LIN {X 0,Y 466.491,Z 652.582,A -85,B 0,C 180,E1 -7510.377,E2 -7510.377} C_VEL
LIN {X 0,Y 466.525,Z 652.204,A -85,B 0,C 180,E1 -7511.517,E2 -7511.517} C_VEL
LIN {X 0,Y 466.577,Z 651.333,A -85,B 0,C 180,E1 -7512.674,E2 -7512.674} C_VEL
LIN {X 0,Y 466.638,Z 649.94,A -85,B 0,C 180,E1 -7513.852,E2 -7513.852} C_VEL
LIN {X 0,Y 466.788,Z 646.773,A -85,B 0,C 180,E1 -7515.615,E2 -7515.615} C_VEL
LIN {X 0,Y 466.978,Z 641.957,A -85,B 0,C 180,E1 -7517.514,E2 -7517.514} C_VEL
LIN {X 0,Y 467.197,Z 636.151,A -85,B 0,C 180,E1 -7519.246,E2 -7519.246} C_VEL
LIN {X 0,Y 467.651,Z 629.363,A -85,B 0,C 180,E1 -7520.861,E2 -7520.861} C_VEL
LIN {X 0,Y 468.11,Z 621.588,A -85,B 0,C 180,E1 -7522.389,E2 -7522.389} C_VEL
LIN {X 0,Y 468.72,Z 612.47,A -85,B 0,C 180,E1 -7523.882,E2 -7523.882} C_VEL
LIN {X 0,Y 469.512,Z 601.824,A -85,B 0,C 180,E1 -7525.332,E2 -7525.332} C_VEL
LIN {X 0,Y 470.362,Z 590.164,A -85,B 0,C 180,E1 -7526.653,E2 -7526.653} C_VEL
LIN {X 0,Y 471.18,Z 578.051,A -85,B 0,C 180,E1 -7527.796,E2 -7527.796} C_VEL
LIN {X 0,Y 472.008,Z 565.223,A -85,B 0,C 180,E1 -7528.797,E2 -7528.797} C_VEL
LIN {X 0,Y 472.783,Z 551.153,A -85,B 0,C 180,E1 -7529.687,E2 -7529.687} C_VEL
LIN {X 0,Y 473.449,Z 536.973,A -85,B 0,C 180,E1 -7530.392,E2 -7530.392} C_VEL
LIN {X 0,Y 473.761,Z 524.414,A -85,B 0,C 180,E1 -7530.885,E2 -7530.885} C_VEL
LIN {X 0,Y 471.201,Z 515.269,A -85,B 0,C 180,E1 -7531.292,E2 -7531.292} C_VEL
LIN {X 0,Y 467.058,Z 503.621,A -85,B 0,C 180,E1 -7531.767,E2 -7531.767} C_VEL
LIN {X 0,Y 466.908,Z 502.739,A -85,B 0,C 180,E1 -7531.818,E2 -7531.818} C_VEL
LIN {X 0,Y 467.035,Z 499.956,A -85,B 0,C 180,E1 -7535.08,E2 -7535.08} C_VEL
LIN {X 0,Y 467.083,Z 497.603,A -85,B 0,C 180,E1 -7537.903,E2 -7537.903} C_VEL
LIN {X 0,Y 467.194,Z 495.312,A -85,B 0,C 180,E1 -7540.673,E2 -7540.673} C_VEL
LIN {X 0,Y 467.284,Z 493.077,A -85,B 0,C 180,E1 -7543.395,E2 -7543.395} C_VEL
LIN {X 0,Y 467.325,Z 490.903,A -85,B 0,C 180,E1 -7546.076,E2 -7546.076} C_VEL
LIN {X 0,Y 467.611,Z 490.865,A -85,B 0,C 180,E1 -7548.732,E2 -7548.732} C_VEL
LIN {X 0,Y 467.746,Z 490.849,A -85,B 0,C 180,E1 -7552.228,E2 -7552.228} C_VEL
LIN {X 0,Y 467.724,Z 490.847,A -85,B 0,C 180,E1 -7554.827,E2 -7554.827} C_VEL
LIN {X 0,Y 467.857,Z 490.832,A -85,B 0,C 180,E1 -7557.417,E2 -7557.417} C_VEL
LIN {X 0,Y 467.878,Z 490.83,A -85,B 0,C 180,E1 -7560,E2 -7560} C_VEL
LIN {X 0,Y 467.856,Z 490.83,A -85,B 0,C 180,E1 -7562.583,E2 -7562.583} C_VEL
LIN {X 0,Y 467.744,Z 490.844,A -85,B 0,C 180,E1 -7566.037,E2 -7566.037} C_VEL
LIN {X 0,Y 467.678,Z 490.854,A -85,B 0,C 180,E1 -7568.643,E2 -7568.643} C_VEL
LIN {X 0,Y 467.653,Z 490.855,A -85,B 0,C 180,E1 -7572.145,E2 -7572.145} C_VEL
LIN {X 0,Y 467.635,Z 490.856,A -85,B 0,C 180,E1 -7575.695,E2 -7575.695} C_VEL
LIN {X 0,Y 467.614,Z 490.863,A -85,B 0,C 180,E1 -7578.765,E2 -7578.765} C_VEL
LIN {X 0,Y 467.577,Z 490.863,A -85,B 0,C 180,E1 -7581.268,E2 -7581.268} C_VEL
LIN {X 0,Y 467.57,Z 490.867,A -85,B 0,C 180,E1 -7583.943,E2 -7583.943} C_VEL
LIN {X 0,Y 467.624,Z 490.86,A -85,B 0,C 180,E1 -7586.8,E2 -7586.8} C_VEL
LIN {X 0,Y 467.584,Z 490.869,A -85,B 0,C 180,E1 -7589.736,E2 -7589.736} C_VEL
LIN {X 0,Y 467.581,Z 490.865,A -85,B 0,C 180,E1 -7592.758,E2 -7592.758} C_VEL
LIN {X 0,Y 467.554,Z 490.871,A -85,B 0,C 180,E1 -7595.889,E2 -7595.889} C_VEL
LIN {X 0,Y 467.579,Z 490.86,A -85,B 0,C 180,E1 -7599.145,E2 -7599.145} C_VEL
LIN {X 0,Y 467.599,Z 490.938,A -85,B 0,C 180,E1 -7602.267,E2 -7602.267} C_VEL
LIN {X 0,Y 468.484,Z 495.805,A -85,B 0,C 180,E1 -7605.165,E2 -7605.165} C_VEL
LIN {X 0,Y 469.206,Z 500.309,A -85,B 0,C 180,E1 -7607.621,E2 -7607.621} C_VEL
LIN {X 0,Y 469.155,Z 504.914,A -85,B 0,C 180,E1 -7609.899,E2 -7609.899} C_VEL
LIN {X 0,Y 468.717,Z 512.053,A -85,B 0,C 180,E1 -7613.147,E2 -7613.147} C_VEL
LIN {X 0,Y 468.459,Z 517.739,A -85,B 0,C 180,E1 -7615.601,E2 -7615.601} C_VEL
LIN {X 0,Y 468.157,Z 525.634,A -85,B 0,C 180,E1 -7618.835,E2 -7618.835} C_VEL
LIN {X 0,Y 467.78,Z 534.355,A -85,B 0,C 180,E1 -7622.241,E2 -7622.241} C_VEL
LIN {X 0,Y 467.603,Z 540.074,A -85,B 0,C 180,E1 -7624.394,E2 -7624.394} C_VEL
LIN {X 0,Y 467.385,Z 548.37,A -85,B 0,C 180,E1 -7627.453,E2 -7627.453} C_VEL
LIN {X 0,Y 467.349,Z 550.449,A -85,B 0,C 180,E1 -7628.204,E2 -7628.204} C_VEL
LIN {X 0,Y 471.32,Z 568.781,A -85,B 0,C 180,E1 -7628.795,E2 -7628.795} C_VEL
LIN {X 0,Y 473.467,Z 579.839,A -85,B 0,C 180,E1 -7629.253,E2 -7629.253} C_VEL
LIN {X 0,Y 472.829,Z 593.635,A -85,B 0,C 180,E1 -7629.807,E2 -7629.807} C_VEL
LIN {X 0,Y 472.025,Z 607.742,A -85,B 0,C 180,E1 -7630.54,E2 -7630.54} C_VEL
LIN {X 0,Y 471.223,Z 621.099,A -85,B 0,C 180,E1 -7631.41,E2 -7631.41} C_VEL
LIN {X 0,Y 470.317,Z 634.718,A -85,B 0,C 180,E1 -7632.498,E2 -7632.498} C_VEL
LIN {X 0,Y 469.526,Z 647.142,A -85,B 0,C 180,E1 -7633.701,E2 -7633.701} C_VEL
LIN {X 0,Y 468.759,Z 658.493,A -85,B 0,C 180,E1 -7635.011,E2 -7635.011} C_VEL
LIN {X 0,Y 468.082,Z 669.532,A -85,B 0,C 180,E1 -7636.542,E2 -7636.542} C_VEL
LIN {X 0,Y 467.594,Z 678.728,A -85,B 0,C 180,E1 -7638.073,E2 -7638.073} C_VEL
LIN {X 0,Y 467.244,Z 686.36,A -85,B 0,C 180,E1 -7639.601,E2 -7639.601} C_VEL
LIN {X 0,Y 466.954,Z 693.49,A -85,B 0,C 180,E1 -7641.343,E2 -7641.343} C_VEL
LIN {X 0,Y 466.819,Z 699.104,A -85,B 0,C 180,E1 -7643.082,E2 -7643.082} C_VEL
LIN {X 0,Y 466.718,Z 703.349,A -85,B 0,C 180,E1 -7644.816,E2 -7644.816} C_VEL
LIN {X 0,Y 466.724,Z 706.332,A -85,B 0,C 180,E1 -7646.546,E2 -7646.546} C_VEL
LIN {X 0,Y 466.681,Z 708.117,A -85,B 0,C 180,E1 -7648.274,E2 -7648.274} C_VEL
LIN {X 0,Y 466.595,Z 708.733,A -85,B 0,C 180,E1 -7650,E2 -7650} C_VEL
LIN {X 0,Y 466.681,Z 708.143,A -85,B 0,C 180,E1 -7651.725,E2 -7651.725} C_VEL
LIN {X 0,Y 466.705,Z 706.385,A -85,B 0,C 180,E1 -7653.453,E2 -7653.453} C_VEL
LIN {X 0,Y 466.717,Z 703.435,A -85,B 0,C 180,E1 -7655.183,E2 -7655.183} C_VEL
LIN {X 0,Y 466.816,Z 699.23,A -85,B 0,C 180,E1 -7656.917,E2 -7656.917} C_VEL
LIN {X 0,Y 466.953,Z 693.655,A -85,B 0,C 180,E1 -7658.656,E2 -7658.656} C_VEL
LIN {X 0,Y 467.243,Z 686.564,A -85,B 0,C 180,E1 -7660.398,E2 -7660.398} C_VEL
LIN {X 0,Y 467.584,Z 678.984,A -85,B 0,C 180,E1 -7661.927,E2 -7661.927} C_VEL
LIN {X 0,Y 468.089,Z 669.852,A -85,B 0,C 180,E1 -7663.457,E2 -7663.457} C_VEL
LIN {X 0,Y 468.792,Z 658.879,A -85,B 0,C 180,E1 -7664.987,E2 -7664.987} C_VEL
LIN {X 0,Y 469.6,Z 647.602,A -85,B 0,C 180,E1 -7666.296,E2 -7666.296} C_VEL
LIN {X 0,Y 470.395,Z 635.248,A -85,B 0,C 180,E1 -7667.498,E2 -7667.498} C_VEL
LIN {X 0,Y 471.333,Z 621.682,A -85,B 0,C 180,E1 -7668.585,E2 -7668.585} C_VEL
LIN {X 0,Y 472.069,Z 608.368,A -85,B 0,C 180,E1 -7669.457,E2 -7669.457} C_VEL
LIN {X 0,Y 472.884,Z 594.139,A -85,B 0,C 180,E1 -7670.199,E2 -7670.199} C_VEL
LIN {X 0,Y 473.519,Z 579.066,A -85,B 0,C 180,E1 -7670.8,E2 -7670.8} C_VEL
LIN {X 0,Y 470.319,Z 564.07,A -85,B 0,C 180,E1 -7671.388,E2 -7671.388} C_VEL
LIN {X 0,Y 467.41,Z 551.33,A -85,B 0,C 180,E1 -7671.791,E2 -7671.791} C_VEL
LIN {X 0,Y 467.633,Z 542.996,A -85,B 0,C 180,E1 -7674.885,E2 -7674.885} C_VEL
LIN {X 0,Y 467.969,Z 534.203,A -85,B 0,C 180,E1 -7678.233,E2 -7678.233} C_VEL
LIN {X 0,Y 468.238,Z 526.736,A -85,B 0,C 180,E1 -7681.181,E2 -7681.181} C_VEL
LIN {X 0,Y 468.555,Z 520.535,A -85,B 0,C 180,E1 -7683.708,E2 -7683.708} C_VEL
LIN {X 0,Y 468.964,Z 511.804,A -85,B 0,C 180,E1 -7687.414,E2 -7687.414} C_VEL
LIN {X 0,Y 469.354,Z 505.502,A -85,B 0,C 180,E1 -7690.212,E2 -7690.212} C_VEL
LIN {X 0,Y 469.457,Z 502.646,A -85,B 0,C 180,E1 -7691.538,E2 -7691.538} C_VEL
LIN {X 0,Y 468.984,Z 498.492,A -85,B 0,C 180,E1 -7693.576,E2 -7693.576} C_VEL
LIN {X 0,Y 468.021,Z 493.263,A -85,B 0,C 180,E1 -7696.31,E2 -7696.31} C_VEL
LIN {X 0,Y 467.608,Z 490.865,A -85,B 0,C 180,E1 -7697.661,E2 -7697.661} C_VEL
LIN {X 0,Y 467.616,Z 490.865,A -85,B 0,C 180,E1 -7700.859,E2 -7700.859} C_VEL
LIN {X 0,Y 467.554,Z 490.871,A -85,B 0,C 180,E1 -7704.26,E2 -7704.26} C_VEL
LIN {X 0,Y 467.573,Z 490.869,A -85,B 0,C 180,E1 -7707.32,E2 -7707.32} C_VEL
LIN {X 0,Y 467.569,Z 490.867,A -85,B 0,C 180,E1 -7710.665,E2 -7710.665} C_VEL
LIN {X 0,Y 467.618,Z 490.864,A -85,B 0,C 180,E1 -7713.2,E2 -7713.2} C_VEL
LIN {X 0,Y 467.582,Z 490.866,A -85,B 0,C 180,E1 -7716.468,E2 -7716.468} C_VEL
LIN {X 0,Y 467.614,Z 490.864,A -85,B 0,C 180,E1 -7719.777,E2 -7719.777} C_VEL
LIN {X 0,Y 467.599,Z 490.863,A -85,B 0,C 180,E1 -7722.507,E2 -7722.507} C_VEL
LIN {X 0,Y 467.596,Z 490.866,A -85,B 0,C 180,E1 -7725.196,E2 -7725.196} C_VEL
LIN {X 0,Y 467.672,Z 490.856,A -85,B 0,C 180,E1 -7727.855,E2 -7727.855} C_VEL
LIN {X 0,Y 467.673,Z 490.857,A -85,B 0,C 180,E1 -7731.357,E2 -7731.357} C_VEL
LIN {X 0,Y 467.738,Z 490.848,A -85,B 0,C 180,E1 -7733.963,E2 -7733.963} C_VEL
LIN {X 0,Y 467.852,Z 490.836,A -85,B 0,C 180,E1 -7737.417,E2 -7737.417} C_VEL
LIN {X 0,Y 467.872,Z 490.831,A -85,B 0,C 180,E1 -7740,E2 -7740} C_VEL
LIN {X 0,Y 467.853,Z 490.832,A -85,B 0,C 180,E1 -7742.583,E2 -7742.583} C_VEL
LIN {X 0,Y 467.745,Z 490.847,A -85,B 0,C 180,E1 -7746.038,E2 -7746.038} C_VEL
LIN {X 0,Y 467.673,Z 490.854,A -85,B 0,C 180,E1 -7748.643,E2 -7748.643} C_VEL
LIN {X 0,Y 467.647,Z 490.859,A -85,B 0,C 180,E1 -7752.146,E2 -7752.146} C_VEL
LIN {X 0,Y 467.63,Z 490.863,A -85,B 0,C 180,E1 -7755.696,E2 -7755.696} C_VEL
LIN {X 0,Y 467.609,Z 490.862,A -85,B 0,C 180,E1 -7758.766,E2 -7758.766} C_VEL
LIN {X 0,Y 467.572,Z 490.869,A -85,B 0,C 180,E1 -7761.269,E2 -7761.269} C_VEL
LIN {X 0,Y 467.565,Z 490.869,A -85,B 0,C 180,E1 -7763.944,E2 -7763.944} C_VEL
LIN {X 0,Y 467.62,Z 490.861,A -85,B 0,C 180,E1 -7766.801,E2 -7766.801} C_VEL
LIN {X 0,Y 467.581,Z 490.868,A -85,B 0,C 180,E1 -7769.737,E2 -7769.737} C_VEL
LIN {X 0,Y 467.578,Z 490.867,A -85,B 0,C 180,E1 -7772.759,E2 -7772.759} C_VEL
LIN {X 0,Y 467.551,Z 490.872,A -85,B 0,C 180,E1 -7775.89,E2 -7775.89} C_VEL
LIN {X 0,Y 467.619,Z 490.863,A -85,B 0,C 180,E1 -7779.142,E2 -7779.142} C_VEL
LIN {X 0,Y 467.615,Z 490.862,A -85,B 0,C 180,E1 -7782.573,E2 -7782.573} C_VEL
LIN {X 0,Y 467.571,Z 490.868,A -85,B 0,C 180,E1 -7786.178,E2 -7786.178} C_VEL
LIN {X 0,Y 467.588,Z 490.864,A -85,B 0,C 180,E1 -7788.723,E2 -7788.723} C_VEL
LIN {X 0,Y 467.577,Z 490.87,A -85,B 0,C 180,E1 -7791.408,E2 -7791.408} C_VEL
LIN {X 0,Y 467.562,Z 490.869,A -85,B 0,C 180,E1 -7794.262,E2 -7794.262} C_VEL
LIN {X 0,Y 467.582,Z 490.868,A -85,B 0,C 180,E1 -7797.322,E2 -7797.322} C_VEL
LIN {X 0,Y 467.571,Z 490.866,A -85,B 0,C 180,E1 -7800.668,E2 -7800.668} C_VEL
LIN {X 0,Y 467.63,Z 490.861,A -85,B 0,C 180,E1 -7803.202,E2 -7803.202} C_VEL
LIN {X 0,Y 467.595,Z 490.864,A -85,B 0,C 180,E1 -7806.469,E2 -7806.469} C_VEL
LIN {X 0,Y 467.626,Z 490.864,A -85,B 0,C 180,E1 -7809.778,E2 -7809.778} C_VEL
LIN {X 0,Y 467.613,Z 490.861,A -85,B 0,C 180,E1 -7812.508,E2 -7812.508} C_VEL
LIN {X 0,Y 467.601,Z 490.864,A -85,B 0,C 180,E1 -7815.434,E2 -7815.434} C_VEL
LIN {X 0,Y 466.931,Z 490.949,A -85,B 0,C 180,E1 -7816.153,E2 -7816.153} C_VEL
LIN {X 0,Y 464.087,Z 491.303,A -85,B 0,C 180,E1 -7817.322,E2 -7817.322} C_VEL
LIN {X 0,Y 461.687,Z 491.601,A -85,B 0,C 180,E1 -7818.264,E2 -7818.264} C_VEL
LIN {X 0,Y 460.66,Z 491.729,A -85,B 0,C 180,E1 -7818.991,E2 -7818.991} C_VEL
LIN {X 0,Y 460.578,Z 491.739,A -85,B 0,C 180,E1 -7819.238,E2 -7819.238} C_VEL
LIN {X 0,Y 460.693,Z 491.723,A -85,B 0,C 180,E1 -7822.57,E2 -7822.57} C_VEL
LIN {X 0,Y 460.703,Z 491.722,A -85,B 0,C 180,E1 -7824.749,E2 -7824.749} C_VEL
LIN {X 0,Y 460.83,Z 491.709,A -85,B 0,C 180,E1 -7827.378,E2 -7827.378} C_VEL
LIN {X 0,Y 460.858,Z 491.705,A -85,B 0,C 180,E1 -7830,E2 -7830} C_VEL
LIN {X 0,Y 460.594,Z 491.737,A -85,B 0,C 180,E1 -7832.624,E2 -7832.624} C_VEL
LIN {X 0,Y 460.297,Z 491.777,A -85,B 0,C 180,E1 -7835.257,E2 -7835.257} C_VEL
LIN {X 0,Y 460.121,Z 491.799,A -85,B 0,C 180,E1 -7836.138,E2 -7836.138} C_VEL
LIN {X 0,Y 460.102,Z 493.135,A -85,B 0,C 180,E1 -7837.902,E2 -7837.902} C_VEL
LIN {X 0,Y 460.014,Z 496.292,A -85,B 0,C 180,E1 -7841.456,E2 -7841.456} C_VEL
LIN {X 0,Y 459.909,Z 498.711,A -85,B 0,C 180,E1 -7844.152,E2 -7844.152} C_VEL
LIN {X 0,Y 459.833,Z 501.178,A -85,B 0,C 180,E1 -7846.882,E2 -7846.882} C_VEL
LIN {X 0,Y 459.829,Z 502.137,A -85,B 0,C 180,E1 -7847.937,E2 -7847.937} C_VEL
LIN {X 0,Y 461.465,Z 507.347,A -85,B 0,C 180,E1 -7848.146,E2 -7848.146} C_VEL
LIN {X 0,Y 466.199,Z 522.117,A -85,B 0,C 180,E1 -7848.791,E2 -7848.791} C_VEL
LIN {X 0,Y 467.154,Z 527.522,A -85,B 0,C 180,E1 -7849.032,E2 -7849.032} C_VEL
LIN {X 0,Y 466.486,Z 542.267,A -85,B 0,C 180,E1 -7849.656,E2 -7849.656} C_VEL
LIN {X 0,Y 465.662,Z 557.391,A -85,B 0,C 180,E1 -7850.499,E2 -7850.499} C_VEL
LIN {X 0,Y 464.865,Z 570.16,A -85,B 0,C 180,E1 -7851.391,E2 -7851.391} C_VEL
LIN {X 0,Y 464.098,Z 581.875,A -85,B 0,C 180,E1 -7852.378,E2 -7852.378} C_VEL
LIN {X 0,Y 463.162,Z 593.929,A -85,B 0,C 180,E1 -7853.591,E2 -7853.591} C_VEL
LIN {X 0,Y 462.346,Z 604.968,A -85,B 0,C 180,E1 -7854.926,E2 -7854.926} C_VEL
LIN {X 0,Y 461.592,Z 615.436,A -85,B 0,C 180,E1 -7856.446,E2 -7856.446} C_VEL
LIN {X 0,Y 461.007,Z 623.526,A -85,B 0,C 180,E1 -7857.845,E2 -7857.845} C_VEL
LIN {X 0,Y 460.468,Z 631.686,A -85,B 0,C 180,E1 -7859.543,E2 -7859.543} C_VEL
LIN {X 0,Y 460.087,Z 638.469,A -85,B 0,C 180,E1 -7861.289,E2 -7861.289} C_VEL
LIN {X 0,Y 459.855,Z 643.153,A -85,B 0,C 180,E1 -7862.799,E2 -7862.799} C_VEL
LIN {X 0,Y 459.702,Z 647.189,A -85,B 0,C 180,E1 -7864.448,E2 -7864.448} C_VEL
LIN {X 0,Y 459.529,Z 649.752,A -85,B 0,C 180,E1 -7865.847,E2 -7865.847} C_VEL
LIN {X 0,Y 459.456,Z 652.014,A -85,B 0,C 180,E1 -7867.723,E2 -7867.723} C_VEL
LIN {X 0,Y 459.446,Z 652.757,A -85,B 0,C 180,E1 -7868.841,E2 -7868.841} C_VEL
LIN {X 0,Y 459.408,Z 653.058,A -85,B 0,C 180,E1 -7870.101,E2 -7870.101} C_VEL
LIN {X 0,Y 459.437,Z 652.681,A -85,B 0,C 180,E1 -7871.448,E2 -7871.448} C_VEL
LIN {X 0,Y 459.507,Z 651.719,A -85,B 0,C 180,E1 -7872.764,E2 -7872.764} C_VEL
LIN {X 0,Y 459.61,Z 649.116,A -85,B 0,C 180,E1 -7874.7,E2 -7874.7} C_VEL
LIN {X 0,Y 459.799,Z 645.282,A -85,B 0,C 180,E1 -7876.541,E2 -7876.541} C_VEL
LIN {X 0,Y 460.021,Z 640.793,A -85,B 0,C 180,E1 -7878.149,E2 -7878.149} C_VEL
LIN {X 0,Y 460.286,Z 635.133,A -85,B 0,C 180,E1 -7879.768,E2 -7879.768} C_VEL
LIN {X 0,Y 460.697,Z 628.659,A -85,B 0,C 180,E1 -7881.283,E2 -7881.283} C_VEL
LIN {X 0,Y 461.331,Z 619.665,A -85,B 0,C 180,E1 -7883.004,E2 -7883.004} C_VEL
LIN {X 0,Y 461.987,Z 610.452,A -85,B 0,C 180,E1 -7884.465,E2 -7884.465} C_VEL
LIN {X 0,Y 462.822,Z 600.26,A -85,B 0,C 180,E1 -7885.816,E2 -7885.816} C_VEL
LIN {X 0,Y 463.639,Z 589.154,A -85,B 0,C 180,E1 -7887.057,E2 -7887.057} C_VEL
LIN {X 0,Y 464.497,Z 577.465,A -85,B 0,C 180,E1 -7888.151,E2 -7888.151} C_VEL
LIN {X 0,Y 465.314,Z 565.338,A -85,B 0,C 180,E1 -7889.1,E2 -7889.1} C_VEL
LIN {X 0,Y 466.128,Z 551.519,A -85,B 0,C 180,E1 -7889.983,E2 -7889.983} C_VEL
LIN {X 0,Y 466.839,Z 537.294,A -85,B 0,C 180,E1 -7890.698,E2 -7890.698} C_VEL
LIN {X 0,Y 467.137,Z 525.812,A -85,B 0,C 180,E1 -7891.159,E2 -7891.159} C_VEL
LIN {X 0,Y 464.156,Z 515.656,A -85,B 0,C 180,E1 -7891.636,E2 -7891.636} C_VEL
LIN {X 0,Y 459.868,Z 503.238,A -85,B 0,C 180,E1 -7892.165,E2 -7892.165} C_VEL
LIN {X 0,Y 459.963,Z 501.123,A -85,B 0,C 180,E1 -7894.67,E2 -7894.67} C_VEL
LIN {X 0,Y 460.028,Z 498.738,A -85,B 0,C 180,E1 -7897.546,E2 -7897.546} C_VEL
LIN {X 0,Y 460.118,Z 496.435,A -85,B 0,C 180,E1 -7900.364,E2 -7900.364} C_VEL
LIN {X 0,Y 460.217,Z 494.172,A -85,B 0,C 180,E1 -7903.133,E2 -7903.133} C_VEL
LIN {X 0,Y 460.28,Z 491.986,A -85,B 0,C 180,E1 -7905.859,E2 -7905.859} C_VEL
LIN {X 0,Y 460.557,Z 491.745,A -85,B 0,C 180,E1 -7908.558,E2 -7908.558} C_VEL
LIN {X 0,Y 460.626,Z 491.732,A -85,B 0,C 180,E1 -7911.223,E2 -7911.223} C_VEL
LIN {X 0,Y 460.708,Z 491.726,A -85,B 0,C 180,E1 -7913.87,E2 -7913.87} C_VEL
LIN {X 0,Y 460.822,Z 491.708,A -85,B 0,C 180,E1 -7917.377,E2 -7917.377} C_VEL
LIN {X 0,Y 460.849,Z 491.706,A -85,B 0,C 180,E1 -7920,E2 -7920} C_VEL
LIN {X 0,Y 460.821,Z 491.707,A -85,B 0,C 180,E1 -7922.622,E2 -7922.622} C_VEL
LIN {X 0,Y 460.709,Z 491.72,A -85,B 0,C 180,E1 -7926.13,E2 -7926.13} C_VEL
LIN {X 0,Y 460.625,Z 491.734,A -85,B 0,C 180,E1 -7928.776,E2 -7928.776} C_VEL
LIN {X 0,Y 460.609,Z 491.734,A -85,B 0,C 180,E1 -7932.445,E2 -7932.445} C_VEL
LIN {X 0,Y 460.596,Z 491.733,A -85,B 0,C 180,E1 -7935.997,E2 -7935.997} C_VEL
LIN {X 0,Y 460.567,Z 491.739,A -85,B 0,C 180,E1 -7938.902,E2 -7938.902} C_VEL
LIN {X 0,Y 460.512,Z 491.743,A -85,B 0,C 180,E1 -7941.485,E2 -7941.485} C_VEL
LIN {X 0,Y 460.539,Z 491.746,A -85,B 0,C 180,E1 -7944.332,E2 -7944.332} C_VEL
LIN {X 0,Y 460.58,Z 491.736,A -85,B 0,C 180,E1 -7947.243,E2 -7947.243} C_VEL
LIN {X 0,Y 460.524,Z 491.747,A -85,B 0,C 180,E1 -7950.239,E2 -7950.239} C_VEL
LIN {X 0,Y 460.526,Z 491.745,A -85,B 0,C 180,E1 -7953.325,E2 -7953.325} C_VEL
LIN {X 0,Y 460.476,Z 491.752,A -85,B 0,C 180,E1 -7956.529,E2 -7956.529} C_VEL
LIN {X 0,Y 460.542,Z 491.737,A -85,B 0,C 180,E1 -7958.898,E2 -7958.898} C_VEL
LIN {X 0,Y 460.54,Z 491.815,A -85,B 0,C 180,E1 -7961.854,E2 -7961.854} C_VEL
LIN {X 0,Y 461.312,Z 496.089,A -85,B 0,C 180,E1 -7964.491,E2 -7964.491} C_VEL
LIN {X 0,Y 462.21,Z 501.339,A -85,B 0,C 180,E1 -7967.465,E2 -7967.465} C_VEL
LIN {X 0,Y 462.224,Z 505.369,A -85,B 0,C 180,E1 -7969.485,E2 -7969.485} C_VEL
LIN {X 0,Y 461.786,Z 511.771,A -85,B 0,C 180,E1 -7972.5,E2 -7972.5} C_VEL
LIN {X 0,Y 461.467,Z 518.181,A -85,B 0,C 180,E1 -7975.326,E2 -7975.326} C_VEL
LIN {X 0,Y 461.118,Z 526.455,A -85,B 0,C 180,E1 -7978.788,E2 -7978.788} C_VEL
LIN {X 0,Y 460.733,Z 535.085,A -85,B 0,C 180,E1 -7982.218,E2 -7982.218} C_VEL
LIN {X 0,Y 460.489,Z 541.544,A -85,B 0,C 180,E1 -7984.701,E2 -7984.701} C_VEL
LIN {X 0,Y 460.288,Z 549.959,A -85,B 0,C 180,E1 -7987.848,E2 -7987.848} C_VEL
LIN {X 0,Y 464.082,Z 567.356,A -85,B 0,C 180,E1 -7988.424,E2 -7988.424} C_VEL
LIN {X 0,Y 466.744,Z 580.449,A -85,B 0,C 180,E1 -7988.982,E2 -7988.982} C_VEL
LIN {X 0,Y 466.081,Z 593.569,A -85,B 0,C 180,E1 -7989.524,E2 -7989.524} C_VEL
LIN {X 0,Y 465.29,Z 607.238,A -85,B 0,C 180,E1 -7990.247,E2 -7990.247} C_VEL
LIN {X 0,Y 464.444,Z 620.597,A -85,B 0,C 180,E1 -7991.128,E2 -7991.128} C_VEL
LIN {X 0,Y 463.472,Z 634.221,A -85,B 0,C 180,E1 -7992.231,E2 -7992.231} C_VEL
LIN {X 0,Y 462.655,Z 646.65,A -85,B 0,C 180,E1 -7993.452,E2 -7993.452} C_VEL
LIN {X 0,Y 461.814,Z 658,A -85,B 0,C 180,E1 -7994.781,E2 -7994.781} C_VEL
LIN {X 0,Y 461.095,Z 669.045,A -85,B 0,C 180,E1 -7996.334,E2 -7996.334} C_VEL
LIN {X 0,Y 460.535,Z 678.247,A -85,B 0,C 180,E1 -7997.887,E2 -7997.887} C_VEL
LIN {X 0,Y 460.175,Z 685.89,A -85,B 0,C 180,E1 -7999.439,E2 -7999.439} C_VEL
LIN {X 0,Y 459.888,Z 693.032,A -85,B 0,C 180,E1 -8001.209,E2 -8001.209} C_VEL
LIN {X 0,Y 459.729,Z 698.654,A -85,B 0,C 180,E1 -8002.975,E2 -8002.975} C_VEL
LIN {X 0,Y 459.626,Z 702.908,A -85,B 0,C 180,E1 -8004.736,E2 -8004.736} C_VEL
LIN {X 0,Y 459.633,Z 705.898,A -85,B 0,C 180,E1 -8006.493,E2 -8006.493} C_VEL
LIN {X 0,Y 459.616,Z 707.688,A -85,B 0,C 180,E1 -8008.247,E2 -8008.247} C_VEL
LIN {X 0,Y 459.527,Z 708.309,A -85,B 0,C 180,E1 -8010,E2 -8010} C_VEL
LIN {X 0,Y 459.616,Z 707.721,A -85,B 0,C 180,E1 -8011.752,E2 -8011.752} C_VEL
LIN {X 0,Y 459.617,Z 705.963,A -85,B 0,C 180,E1 -8013.506,E2 -8013.506} C_VEL
LIN {X 0,Y 459.626,Z 703.013,A -85,B 0,C 180,E1 -8015.263,E2 -8015.263} C_VEL
LIN {X 0,Y 459.727,Z 698.806,A -85,B 0,C 180,E1 -8017.024,E2 -8017.024} C_VEL
LIN {X 0,Y 459.887,Z 693.229,A -85,B 0,C 180,E1 -8018.79,E2 -8018.79} C_VEL
LIN {X 0,Y 460.173,Z 686.135,A -85,B 0,C 180,E1 -8020.56,E2 -8020.56} C_VEL
LIN {X 0,Y 460.536,Z 678.552,A -85,B 0,C 180,E1 -8022.112,E2 -8022.112} C_VEL
LIN {X 0,Y 461.103,Z 669.419,A -85,B 0,C 180,E1 -8023.664,E2 -8023.664} C_VEL
LIN {X 0,Y 461.828,Z 658.44,A -85,B 0,C 180,E1 -8025.218,E2 -8025.218} C_VEL
LIN {X 0,Y 462.697,Z 647.161,A -85,B 0,C 180,E1 -8026.546,E2 -8026.546} C_VEL
LIN {X 0,Y 463.534,Z 634.802,A -85,B 0,C 180,E1 -8027.765,E2 -8027.765} C_VEL
LIN {X 0,Y 464.525,Z 621.222,A -85,B 0,C 180,E1 -8028.867,E2 -8028.867} C_VEL
LIN {X 0,Y 465.35,Z 607.898,A -85,B 0,C 180,E1 -8029.749,E2 -8029.749} C_VEL
LIN {X 0,Y 466.167,Z 594.09,A -85,B 0,C 180,E1 -8030.48,E2 -8030.48} C_VEL
LIN {X 0,Y 466.68,Z 579.68,A -85,B 0,C 180,E1 -8031.076,E2 -8031.076} C_VEL
LIN {X 0,Y 463.342,Z 563.977,A -85,B 0,C 180,E1 -8031.713,E2 -8031.713} C_VEL
LIN {X 0,Y 460.364,Z 550.917,A -85,B 0,C 180,E1 -8032.141,E2 -8032.141} C_VEL
LIN {X 0,Y 460.623,Z 542.565,A -85,B 0,C 180,E1 -8035.29,E2 -8035.29} C_VEL
LIN {X 0,Y 460.958,Z 533.877,A -85,B 0,C 180,E1 -8038.702,E2 -8038.702} C_VEL
LIN {X 0,Y 461.264,Z 527.064,A -85,B 0,C 180,E1 -8041.435,E2 -8041.435} C_VEL
LIN {X 0,Y 461.577,Z 520.241,A -85,B 0,C 180,E1 -8044.287,E2 -8044.287} C_VEL
LIN {X 0,Y 462.007,Z 512.325,A -85,B 0,C 180,E1 -8047.72,E2 -8047.72} C_VEL
LIN {X 0,Y 462.423,Z 505.546,A -85,B 0,C 180,E1 -8050.806,E2 -8050.806} C_VEL
LIN {X 0,Y 462.348,Z 501.938,A -85,B 0,C 180,E1 -8052.536,E2 -8052.536} C_VEL
LIN {X 0,Y 461.349,Z 496.199,A -85,B 0,C 180,E1 -8055.513,E2 -8055.513} C_VEL
LIN {X 0,Y 460.562,Z 491.743,A -85,B 0,C 180,E1 -8057.985,E2 -8057.985} C_VEL
LIN {X 0,Y 460.541,Z 491.745,A -85,B 0,C 180,E1 -8061.269,E2 -8061.269} C_VEL
LIN {X 0,Y 460.505,Z 491.748,A -85,B 0,C 180,E1 -8064.554,E2 -8064.554} C_VEL
LIN {X 0,Y 460.523,Z 491.747,A -85,B 0,C 180,E1 -8067.715,E2 -8067.715} C_VEL
LIN {X 0,Y 460.538,Z 491.743,A -85,B 0,C 180,E1 -8070.769,E2 -8070.769} C_VEL
LIN {X 0,Y 460.558,Z 491.743,A -85,B 0,C 180,E1 -8073.735,E2 -8073.735} C_VEL
LIN {X 0,Y 460.536,Z 491.743,A -85,B 0,C 180,E1 -8076.624,E2 -8076.624} C_VEL
LIN {X 0,Y 460.542,Z 491.746,A -85,B 0,C 180,E1 -8079.453,E2 -8079.453} C_VEL
LIN {X 0,Y 460.549,Z 491.741,A -85,B 0,C 180,E1 -8082.23,E2 -8082.23} C_VEL
LIN {X 0,Y 460.559,Z 491.741,A -85,B 0,C 180,E1 -8084.965,E2 -8084.965} C_VEL
LIN {X 0,Y 460.619,Z 491.736,A -85,B 0,C 180,E1 -8087.666,E2 -8087.666} C_VEL
LIN {X 0,Y 460.62,Z 491.735,A -85,B 0,C 180,E1 -8091.224,E2 -8091.224} C_VEL
LIN {X 0,Y 460.703,Z 491.725,A -85,B 0,C 180,E1 -8093.87,E2 -8093.87} C_VEL
LIN {X 0,Y 460.817,Z 491.712,A -85,B 0,C 180,E1 -8097.378,E2 -8097.378} C_VEL
LIN {X 0,Y 460.843,Z 491.707,A -85,B 0,C 180,E1 -8100,E2 -8100} C_VEL
LIN {X 0,Y 460.818,Z 491.708,A -85,B 0,C 180,E1 -8102.623,E2 -8102.623} C_VEL
LIN {X 0,Y 460.709,Z 491.722,A -85,B 0,C 180,E1 -8106.13,E2 -8106.13} C_VEL
LIN {X 0,Y 460.62,Z 491.733,A -85,B 0,C 180,E1 -8108.777,E2 -8108.777} C_VEL
LIN {X 0,Y 460.603,Z 491.735,A -85,B 0,C 180,E1 -8112.446,E2 -8112.446} C_VEL
LIN {X 0,Y 460.591,Z 491.738,A -85,B 0,C 180,E1 -8115.998,E2 -8115.998} C_VEL
LIN {X 0,Y 460.562,Z 491.74,A -85,B 0,C 180,E1 -8118.903,E2 -8118.903} C_VEL
LIN {X 0,Y 460.508,Z 491.751,A -85,B 0,C 180,E1 -8121.486,E2 -8121.486} C_VEL
LIN {X 0,Y 460.535,Z 491.744,A -85,B 0,C 180,E1 -8124.333,E2 -8124.333} C_VEL
LIN {X 0,Y 460.577,Z 491.741,A -85,B 0,C 180,E1 -8127.244,E2 -8127.244} C_VEL
LIN {X 0,Y 460.52,Z 491.746,A -85,B 0,C 180,E1 -8130.24,E2 -8130.24} C_VEL
LIN {X 0,Y 460.523,Z 491.747,A -85,B 0,C 180,E1 -8133.326,E2 -8133.326} C_VEL
LIN {X 0,Y 460.474,Z 491.751,A -85,B 0,C 180,E1 -8136.53,E2 -8136.53} C_VEL
LIN {X 0,Y 460.58,Z 491.741,A -85,B 0,C 180,E1 -8139.858,E2 -8139.858} C_VEL
LIN {X 0,Y 460.539,Z 491.744,A -85,B 0,C 180,E1 -8142.906,E2 -8142.906} C_VEL
LIN {X 0,Y 460.521,Z 491.748,A -85,B 0,C 180,E1 -8145.83,E2 -8145.83} C_VEL
LIN {X 0,Y 460.541,Z 491.743,A -85,B 0,C 180,E1 -8148.991,E2 -8148.991} C_VEL
LIN {X 0,Y 460.546,Z 491.745,A -85,B 0,C 180,E1 -8151.27,E2 -8151.27} C_VEL
LIN {X 0,Y 460.512,Z 491.746,A -85,B 0,C 180,E1 -8154.556,E2 -8154.556} C_VEL
LIN {X 0,Y 460.532,Z 491.748,A -85,B 0,C 180,E1 -8157.717,E2 -8157.717} C_VEL
LIN {X 0,Y 460.541,Z 491.742,A -85,B 0,C 180,E1 -8160.77,E2 -8160.77} C_VEL
LIN {X 0,Y 460.57,Z 491.742,A -85,B 0,C 180,E1 -8163.736,E2 -8163.736} C_VEL
LIN {X 0,Y 460.549,Z 491.742,A -85,B 0,C 180,E1 -8166.625,E2 -8166.625} C_VEL
LIN {X 0,Y 460.554,Z 491.744,A -85,B 0,C 180,E1 -8169.454,E2 -8169.454} C_VEL
LIN {X 0,Y 460.563,Z 491.74,A -85,B 0,C 180,E1 -8172.231,E2 -8172.231} C_VEL
LIN {X 0,Y 460.57,Z 491.74,A -85,B 0,C 180,E1 -8174.966,E2 -8174.966} C_VEL
LIN {X 0,Y 460.614,Z 491.734,A -85,B 0,C 180,E1 -8178.56,E2 -8178.56} C_VEL
LIN {X 0,Y 460.578,Z 491.739,A -85,B 0,C 180,E1 -8179.238,E2 -8179.238} C_VEL
LIN {X 0,Y 459.919,Z 491.824,A -85,B 0,C 180,E1 -8179.968,E2 -8179.968} C_VEL
LIN {X 0,Y 457.091,Z 492.176,A -85,B 0,C 180,E1 -8181.154,E2 -8181.154} C_VEL
LIN {X 0,Y 454.708,Z 492.47,A -85,B 0,C 180,E1 -8182.11,E2 -8182.11} C_VEL
LIN {X 0,Y 453.7,Z 492.594,A -85,B 0,C 180,E1 -8182.849,E2 -8182.849} C_VEL
LIN {X 0,Y 453.627,Z 492.603,A -85,B 0,C 180,E1 -8183.099,E2 -8183.099} C_VEL
LIN {X 0,Y 453.676,Z 492.597,A -85,B 0,C 180,E1 -8184.667,E2 -8184.667} C_VEL
LIN {X 0,Y 453.771,Z 492.588,A -85,B 0,C 180,E1 -8187.337,E2 -8187.337} C_VEL
LIN {X 0,Y 453.828,Z 492.58,A -85,B 0,C 180,E1 -8190,E2 -8190} C_VEL
LIN {X 0,Y 453.551,Z 492.614,A -85,B 0,C 180,E1 -8192.665,E2 -8192.665} C_VEL
LIN {X 0,Y 453.236,Z 492.656,A -85,B 0,C 180,E1 -8195.339,E2 -8195.339} C_VEL
LIN {X 0,Y 453.069,Z 492.677,A -85,B 0,C 180,E1 -8196.234,E2 -8196.234} C_VEL
LIN {X 0,Y 453.027,Z 493.993,A -85,B 0,C 180,E1 -8198.026,E2 -8198.026} C_VEL
LIN {X 0,Y 452.944,Z 497.175,A -85,B 0,C 180,E1 -8201.637,E2 -8201.637} C_VEL
LIN {X 0,Y 452.833,Z 499.618,A -85,B 0,C 180,E1 -8204.378,E2 -8204.378} C_VEL
LIN {X 0,Y 452.767,Z 502.521,A -85,B 0,C 180,E1 -8207.59,E2 -8207.59} C_VEL
LIN {X 0,Y 455.296,Z 510.287,A -85,B 0,C 180,E1 -8207.895,E2 -8207.895} C_VEL
LIN {X 0,Y 459.894,Z 524.997,A -85,B 0,C 180,E1 -8208.575,E2 -8208.575} C_VEL
LIN {X 0,Y 460.502,Z 528.499,A -85,B 0,C 180,E1 -8208.742,E2 -8208.742} C_VEL
LIN {X 0,Y 459.773,Z 543.95,A -85,B 0,C 180,E1 -8209.418,E2 -8209.418} C_VEL
LIN {X 0,Y 459.036,Z 556.86,A -85,B 0,C 180,E1 -8210.15,E2 -8210.15} C_VEL
LIN {X 0,Y 458.161,Z 570.163,A -85,B 0,C 180,E1 -8211.083,E2 -8211.083} C_VEL
LIN {X 0,Y 457.325,Z 582.306,A -85,B 0,C 180,E1 -8212.118,E2 -8212.118} C_VEL
LIN {X 0,Y 456.317,Z 594.499,A -85,B 0,C 180,E1 -8213.365,E2 -8213.365} C_VEL
LIN {X 0,Y 455.516,Z 604.78,A -85,B 0,C 180,E1 -8214.618,E2 -8214.618} C_VEL
LIN {X 0,Y 454.695,Z 615.537,A -85,B 0,C 180,E1 -8216.191,E2 -8216.191} C_VEL
LIN {X 0,Y 454.031,Z 623.978,A -85,B 0,C 180,E1 -8217.67,E2 -8217.67} C_VEL
LIN {X 0,Y 453.445,Z 632.506,A -85,B 0,C 180,E1 -8219.478,E2 -8219.478} C_VEL
LIN {X 0,Y 453.02,Z 639.799,A -85,B 0,C 180,E1 -8221.432,E2 -8221.432} C_VEL
LIN {X 0,Y 452.77,Z 644.555,A -85,B 0,C 180,E1 -8223.048,E2 -8223.048} C_VEL
LIN {X 0,Y 452.56,Z 649.008,A -85,B 0,C 180,E1 -8225.071,E2 -8225.071} C_VEL
LIN {X 0,Y 452.432,Z 650.769,A -85,B 0,C 180,E1 -8226.177,E2 -8226.177} C_VEL
LIN {X 0,Y 452.378,Z 652.355,A -85,B 0,C 180,E1 -8227.596,E2 -8227.596} C_VEL
LIN {X 0,Y 452.343,Z 653.402,A -85,B 0,C 180,E1 -8229.569,E2 -8229.569} C_VEL
LIN {X 0,Y 452.324,Z 653.382,A -85,B 0,C 180,E1 -8230.736,E2 -8230.736} C_VEL
LIN {X 0,Y 452.354,Z 652.882,A -85,B 0,C 180,E1 -8231.918,E2 -8231.918} C_VEL
LIN {X 0,Y 452.436,Z 651.851,A -85,B 0,C 180,E1 -8233.116,E2 -8233.116} C_VEL
LIN {X 0,Y 452.577,Z 649.258,A -85,B 0,C 180,E1 -8234.955,E2 -8234.955} C_VEL
LIN {X 0,Y 452.798,Z 645.051,A -85,B 0,C 180,E1 -8236.926,E2 -8236.926} C_VEL
LIN {X 0,Y 453.027,Z 639.759,A -85,B 0,C 180,E1 -8238.751,E2 -8238.751} C_VEL
LIN {X 0,Y 453.49,Z 633.077,A -85,B 0,C 180,E1 -8240.55,E2 -8240.55} C_VEL
LIN {X 0,Y 453.973,Z 625.773,A -85,B 0,C 180,E1 -8242.142,E2 -8242.142} C_VEL
LIN {X 0,Y 454.697,Z 616.727,A -85,B 0,C 180,E1 -8243.774,E2 -8243.774} C_VEL
LIN {X 0,Y 455.429,Z 607.376,A -85,B 0,C 180,E1 -8245.182,E2 -8245.182} C_VEL
LIN {X 0,Y 456.345,Z 596.191,A -85,B 0,C 180,E1 -8246.593,E2 -8246.593} C_VEL
LIN {X 0,Y 457.267,Z 584.536,A -85,B 0,C 180,E1 -8247.819,E2 -8247.819} C_VEL
LIN {X 0,Y 458.187,Z 571.801,A -85,B 0,C 180,E1 -8248.935,E2 -8248.935} C_VEL
LIN {X 0,Y 459.089,Z 558.234,A -85,B 0,C 180,E1 -8249.905,E2 -8249.905} C_VEL
LIN {X 0,Y 459.962,Z 543.72,A -85,B 0,C 180,E1 -8250.728,E2 -8250.728} C_VEL
LIN {X 0,Y 460.602,Z 528.438,A -85,B 0,C 180,E1 -8251.392,E2 -8251.392} C_VEL
LIN {X 0,Y 459.381,Z 522.946,A -85,B 0,C 180,E1 -8251.657,E2 -8251.657} C_VEL
LIN {X 0,Y 454.635,Z 509.076,A -85,B 0,C 180,E1 -8252.307,E2 -8252.307} C_VEL
LIN {X 0,Y 452.848,Z 503.731,A -85,B 0,C 180,E1 -8252.534,E2 -8252.534} C_VEL
LIN {X 0,Y 452.913,Z 501.493,A -85,B 0,C 180,E1 -8255.23,E2 -8255.23} C_VEL
LIN {X 0,Y 453.036,Z 498.756,A -85,B 0,C 180,E1 -8258.556,E2 -8258.556} C_VEL
LIN {X 0,Y 453.124,Z 496.035,A -85,B 0,C 180,E1 -8261.928,E2 -8261.928} C_VEL
LIN {X 0,Y 453.243,Z 493.806,A -85,B 0,C 180,E1 -8264.716,E2 -8264.716} C_VEL
LIN {X 0,Y 453.299,Z 492.649,A -85,B 0,C 180,E1 -8266.552,E2 -8266.552} C_VEL
LIN {X 0,Y 453.507,Z 492.621,A -85,B 0,C 180,E1 -8269.282,E2 -8269.282} C_VEL
LIN {X 0,Y 453.689,Z 492.597,A -85,B 0,C 180,E1 -8272.48,E2 -8272.48} C_VEL
LIN {X 0,Y 453.67,Z 492.598,A -85,B 0,C 180,E1 -8274.666,E2 -8274.666} C_VEL
LIN {X 0,Y 453.763,Z 492.587,A -85,B 0,C 180,E1 -8277.336,E2 -8277.336} C_VEL
LIN {X 0,Y 453.82,Z 492.581,A -85,B 0,C 180,E1 -8280,E2 -8280} C_VEL
LIN {X 0,Y 453.761,Z 492.586,A -85,B 0,C 180,E1 -8282.663,E2 -8282.663} C_VEL
LIN {X 0,Y 453.676,Z 492.596,A -85,B 0,C 180,E1 -8286.225,E2 -8286.225} C_VEL
LIN {X 0,Y 453.589,Z 492.611,A -85,B 0,C 180,E1 -8288.913,E2 -8288.913} C_VEL
LIN {X 0,Y 453.559,Z 492.613,A -85,B 0,C 180,E1 -8292.529,E2 -8292.529} C_VEL
LIN {X 0,Y 453.541,Z 492.614,A -85,B 0,C 180,E1 -8296.196,E2 -8296.196} C_VEL
LIN {X 0,Y 453.516,Z 492.617,A -85,B 0,C 180,E1 -8299.041,E2 -8299.041} C_VEL
LIN {X 0,Y 453.473,Z 492.621,A -85,B 0,C 180,E1 -8301.836,E2 -8301.836} C_VEL
LIN {X 0,Y 453.511,Z 492.618,A -85,B 0,C 180,E1 -8304.734,E2 -8304.734} C_VEL
LIN {X 0,Y 453.535,Z 492.619,A -85,B 0,C 180,E1 -8307.961,E2 -8307.961} C_VEL
LIN {X 0,Y 453.48,Z 492.623,A -85,B 0,C 180,E1 -8310.759,E2 -8310.759} C_VEL
LIN {X 0,Y 453.475,Z 492.627,A -85,B 0,C 180,E1 -8313.913,E2 -8313.913} C_VEL
LIN {X 0,Y 453.468,Z 492.625,A -85,B 0,C 180,E1 -8317.188,E2 -8317.188} C_VEL
LIN {X 0,Y 453.487,Z 492.616,A -85,B 0,C 180,E1 -8319.45,E2 -8319.45} C_VEL
LIN {X 0,Y 453.516,Z 492.795,A -85,B 0,C 180,E1 -8321.489,E2 -8321.489} C_VEL
LIN {X 0,Y 454.405,Z 497.821,A -85,B 0,C 180,E1 -8324.647,E2 -8324.647} C_VEL
LIN {X 0,Y 455.171,Z 502.279,A -85,B 0,C 180,E1 -8327.206,E2 -8327.206} C_VEL
LIN {X 0,Y 455.28,Z 505.971,A -85,B 0,C 180,E1 -8329.147,E2 -8329.147} C_VEL
LIN {X 0,Y 454.783,Z 512.915,A -85,B 0,C 180,E1 -8332.468,E2 -8332.468} C_VEL
LIN {X 0,Y 454.48,Z 518.729,A -85,B 0,C 180,E1 -8335.099,E2 -8335.099} C_VEL
LIN {X 0,Y 454.133,Z 526.309,A -85,B 0,C 180,E1 -8338.338,E2 -8338.338} C_VEL
LIN {X 0,Y 453.755,Z 533.556,A -85,B 0,C 180,E1 -8341.305,E2 -8341.305} C_VEL
LIN {X 0,Y 453.487,Z 541.115,A -85,B 0,C 180,E1 -8344.282,E2 -8344.282} C_VEL
LIN {X 0,Y 453.251,Z 549.476,A -85,B 0,C 180,E1 -8347.48,E2 -8347.48} C_VEL
LIN {X 0,Y 457.234,Z 567.252,A -85,B 0,C 180,E1 -8348.09,E2 -8348.09} C_VEL
LIN {X 0,Y 459.971,Z 582.083,A -85,B 0,C 180,E1 -8348.739,E2 -8348.739} C_VEL
LIN {X 0,Y 459.305,Z 595.108,A -85,B 0,C 180,E1 -8349.314,E2 -8349.314} C_VEL
LIN {X 0,Y 458.442,Z 608.507,A -85,B 0,C 180,E1 -8350.056,E2 -8350.056} C_VEL
LIN {X 0,Y 457.549,Z 621.538,A -85,B 0,C 180,E1 -8350.949,E2 -8350.949} C_VEL
LIN {X 0,Y 456.524,Z 634.911,A -85,B 0,C 180,E1 -8352.068,E2 -8352.068} C_VEL
LIN {X 0,Y 455.748,Z 646.157,A -85,B 0,C 180,E1 -8353.193,E2 -8353.193} C_VEL
LIN {X 0,Y 454.872,Z 657.516,A -85,B 0,C 180,E1 -8354.542,E2 -8354.542} C_VEL
LIN {X 0,Y 454.122,Z 668.571,A -85,B 0,C 180,E1 -8356.12,E2 -8356.12} C_VEL
LIN {X 0,Y 453.49,Z 677.622,A -85,B 0,C 180,E1 -8357.668,E2 -8357.668} C_VEL
LIN {X 0,Y 453.136,Z 685.423,A -85,B 0,C 180,E1 -8359.274,E2 -8359.274} C_VEL
LIN {X 0,Y 452.794,Z 692.571,A -85,B 0,C 180,E1 -8361.07,E2 -8361.07} C_VEL
LIN {X 0,Y 452.648,Z 698.205,A -85,B 0,C 180,E1 -8362.864,E2 -8362.864} C_VEL
LIN {X 0,Y 452.538,Z 702.467,A -85,B 0,C 180,E1 -8364.653,E2 -8364.653} C_VEL
LIN {X 0,Y 452.531,Z 705.464,A -85,B 0,C 180,E1 -8366.438,E2 -8366.438} C_VEL
LIN {X 0,Y 452.523,Z 707.258,A -85,B 0,C 180,E1 -8368.22,E2 -8368.22} C_VEL
LIN {X 0,Y 452.461,Z 707.884,A -85,B 0,C 180,E1 -8370,E2 -8370} C_VEL
LIN {X 0,Y 452.523,Z 707.298,A -85,B 0,C 180,E1 -8371.779,E2 -8371.779} C_VEL
LIN {X 0,Y 452.516,Z 705.541,A -85,B 0,C 180,E1 -8373.561,E2 -8373.561} C_VEL
LIN {X 0,Y 452.538,Z 702.592,A -85,B 0,C 180,E1 -8375.346,E2 -8375.346} C_VEL
LIN {X 0,Y 452.646,Z 698.384,A -85,B 0,C 180,E1 -8377.135,E2 -8377.135} C_VEL
LIN {X 0,Y 452.81,Z 692.804,A -85,B 0,C 180,E1 -8378.928,E2 -8378.928} C_VEL
LIN {X 0,Y 453.135,Z 685.708,A -85,B 0,C 180,E1 -8380.726,E2 -8380.726} C_VEL
LIN {X 0,Y 453.512,Z 677.892,A -85,B 0,C 180,E1 -8382.345,E2 -8382.345} C_VEL
LIN {X 0,Y 454.138,Z 668.984,A -85,B 0,C 180,E1 -8383.878,E2 -8383.878} C_VEL
LIN {X 0,Y 454.89,Z 657.991,A -85,B 0,C 180,E1 -8385.456,E2 -8385.456} C_VEL
LIN {X 0,Y 455.77,Z 646.7,A -85,B 0,C 180,E1 -8386.805,E2 -8386.805} C_VEL
LIN {X 0,Y 456.709,Z 634.332,A -85,B 0,C 180,E1 -8388.04,E2 -8388.04} C_VEL
LIN {X 0,Y 457.71,Z 620.736,A -85,B 0,C 180,E1 -8389.159,E2 -8389.159} C_VEL
LIN {X 0,Y 458.618,Z 607.407,A -85,B 0,C 180,E1 -8390.052,E2 -8390.052} C_VEL
LIN {X 0,Y 459.511,Z 592.926,A -85,B 0,C 180,E1 -8390.825,E2 -8390.825} C_VEL
LIN {X 0,Y 459.925,Z 580.617,A -85,B 0,C 180,E1 -8391.344,E2 -8391.344} C_VEL
LIN {X 0,Y 456.533,Z 564.528,A -85,B 0,C 180,E1 -8392.024,E2 -8392.024} C_VEL
LIN {X 0,Y 453.298,Z 550.524,A -85,B 0,C 180,E1 -8392.493,E2 -8392.493} C_VEL
LIN {X 0,Y 453.612,Z 542.229,A -85,B 0,C 180,E1 -8395.709,E2 -8395.709} C_VEL
LIN {X 0,Y 453.898,Z 534.76,A -85,B 0,C 180,E1 -8398.684,E2 -8398.684} C_VEL
LIN {X 0,Y 454.242,Z 527.466,A -85,B 0,C 180,E1 -8401.685,E2 -8401.685} C_VEL
LIN {X 0,Y 454.574,Z 521.168,A -85,B 0,C 180,E1 -8404.353,E2 -8404.353} C_VEL
LIN {X 0,Y 455.043,Z 512.833,A -85,B 0,C 180,E1 -8408.031,E2 -8408.031} C_VEL
LIN {X 0,Y 455.44,Z 506.706,A -85,B 0,C 180,E1 -8410.876,E2 -8410.876} C_VEL
LIN {X 0,Y 455.32,Z 502.837,A -85,B 0,C 180,E1 -8412.776,E2 -8412.776} C_VEL
LIN {X 0,Y 454.271,Z 496.983,A -85,B 0,C 180,E1 -8415.878,E2 -8415.878} C_VEL
LIN {X 0,Y 453.515,Z 492.62,A -85,B 0,C 180,E1 -8418.362,E2 -8418.362} C_VEL
LIN {X 0,Y 453.527,Z 492.619,A -85,B 0,C 180,E1 -8420.786,E2 -8420.786} C_VEL
LIN {X 0,Y 453.449,Z 492.628,A -85,B 0,C 180,E1 -8423.917,E2 -8423.917} C_VEL
LIN {X 0,Y 453.474,Z 492.625,A -85,B 0,C 180,E1 -8427.151,E2 -8427.151} C_VEL
LIN {X 0,Y 453.505,Z 492.619,A -85,B 0,C 180,E1 -8430.271,E2 -8430.271} C_VEL
LIN {X 0,Y 453.504,Z 492.623,A -85,B 0,C 180,E1 -8433.294,E2 -8433.294} C_VEL
LIN {X 0,Y 453.493,Z 492.621,A -85,B 0,C 180,E1 -8436.239,E2 -8436.239} C_VEL
LIN {X 0,Y 453.473,Z 492.625,A -85,B 0,C 180,E1 -8439.117,E2 -8439.117} C_VEL
LIN {X 0,Y 453.502,Z 492.621,A -85,B 0,C 180,E1 -8441.944,E2 -8441.944} C_VEL
LIN {X 0,Y 453.539,Z 492.614,A -85,B 0,C 180,E1 -8444.727,E2 -8444.727} C_VEL
LIN {X 0,Y 453.591,Z 492.612,A -85,B 0,C 180,E1 -8447.472,E2 -8447.472} C_VEL
LIN {X 0,Y 453.584,Z 492.612,A -85,B 0,C 180,E1 -8451.087,E2 -8451.087} C_VEL
LIN {X 0,Y 453.67,Z 492.602,A -85,B 0,C 180,E1 -8453.775,E2 -8453.775} C_VEL
LIN {X 0,Y 453.758,Z 492.591,A -85,B 0,C 180,E1 -8457.337,E2 -8457.337} C_VEL
LIN {X 0,Y 453.814,Z 492.582,A -85,B 0,C 180,E1 -8460,E2 -8460} C_VEL
LIN {X 0,Y 453.758,Z 492.587,A -85,B 0,C 180,E1 -8462.664,E2 -8462.664} C_VEL
LIN {X 0,Y 453.675,Z 492.598,A -85,B 0,C 180,E1 -8466.226,E2 -8466.226} C_VEL
LIN {X 0,Y 453.584,Z 492.61,A -85,B 0,C 180,E1 -8468.914,E2 -8468.914} C_VEL
LIN {X 0,Y 453.554,Z 492.613,A -85,B 0,C 180,E1 -8472.53,E2 -8472.53} C_VEL
LIN {X 0,Y 453.536,Z 492.615,A -85,B 0,C 180,E1 -8476.197,E2 -8476.197} C_VEL
LIN {X 0,Y 453.512,Z 492.619,A -85,B 0,C 180,E1 -8479.042,E2 -8479.042} C_VEL
LIN {X 0,Y 453.468,Z 492.626,A -85,B 0,C 180,E1 -8481.837,E2 -8481.837} C_VEL
LIN {X 0,Y 453.507,Z 492.619,A -85,B 0,C 180,E1 -8484.735,E2 -8484.735} C_VEL
LIN {X 0,Y 453.532,Z 492.618,A -85,B 0,C 180,E1 -8487.962,E2 -8487.962} C_VEL
LIN {X 0,Y 453.477,Z 492.623,A -85,B 0,C 180,E1 -8490.76,E2 -8490.76} C_VEL
LIN {X 0,Y 453.472,Z 492.625,A -85,B 0,C 180,E1 -8493.914,E2 -8493.914} C_VEL
LIN {X 0,Y 453.467,Z 492.626,A -85,B 0,C 180,E1 -8497.189,E2 -8497.189} C_VEL
LIN {X 0,Y 453.532,Z 492.619,A -85,B 0,C 180,E1 -8499.446,E2 -8499.446} C_VEL
LIN {X 0,Y 453.488,Z 492.622,A -85,B 0,C 180,E1 -8502.993,E2 -8502.993} C_VEL
LIN {X 0,Y 453.474,Z 492.626,A -85,B 0,C 180,E1 -8505.782,E2 -8505.782} C_VEL
LIN {X 0,Y 453.494,Z 492.62,A -85,B 0,C 180,E1 -8508.213,E2 -8508.213} C_VEL
LIN {X 0,Y 453.531,Z 492.615,A -85,B 0,C 180,E1 -8510.789,E2 -8510.789} C_VEL
LIN {X 0,Y 453.456,Z 492.627,A -85,B 0,C 180,E1 -8513.919,E2 -8513.919} C_VEL
LIN {X 0,Y 453.483,Z 492.624,A -85,B 0,C 180,E1 -8517.152,E2 -8517.152} C_VEL
LIN {X 0,Y 453.476,Z 492.622,A -85,B 0,C 180,E1 -8520.27,E2 -8520.27} C_VEL
LIN {X 0,Y 453.516,Z 492.62,A -85,B 0,C 180,E1 -8523.296,E2 -8523.296} C_VEL
LIN {X 0,Y 453.506,Z 492.62,A -85,B 0,C 180,E1 -8526.24,E2 -8526.24} C_VEL
LIN {X 0,Y 453.486,Z 492.623,A -85,B 0,C 180,E1 -8529.119,E2 -8529.119} C_VEL
LIN {X 0,Y 453.516,Z 492.621,A -85,B 0,C 180,E1 -8531.946,E2 -8531.946} C_VEL
LIN {X 0,Y 453.544,Z 492.614,A -85,B 0,C 180,E1 -8534.727,E2 -8534.727} C_VEL
LIN {X 0,Y 453.563,Z 492.612,A -85,B 0,C 180,E1 -8538.38,E2 -8538.38} C_VEL
LIN {X 0,Y 453.59,Z 492.61,A -85,B 0,C 180,E1 -8541.087,E2 -8541.087} C_VEL
LIN {X 0,Y 453.627,Z 492.603,A -85,B 0,C 180,E1 -8543.099,E2 -8543.099} C_VEL
LIN {X 0,Y 452.951,Z 492.691,A -85,B 0,C 180,E1 -8543.84,E2 -8543.84} C_VEL
LIN {X 0,Y 450.009,Z 493.055,A -85,B 0,C 180,E1 -8545.041,E2 -8545.041} C_VEL
LIN {X 0,Y 447.587,Z 493.359,A -85,B 0,C 180,E1 -8546.011,E2 -8546.011} C_VEL
LIN {X 0,Y 446.65,Z 493.473,A -85,B 0,C 180,E1 -8546.761,E2 -8546.761} C_VEL
LIN {X 0,Y 446.631,Z 493.475,A -85,B 0,C 180,E1 -8547.015,E2 -8547.015} C_VEL
LIN {X 0,Y 446.798,Z 493.456,A -85,B 0,C 180,E1 -8550,E2 -8550} C_VEL
LIN {X 0,Y 446.509,Z 493.491,A -85,B 0,C 180,E1 -8552.707,E2 -8552.707} C_VEL
LIN {X 0,Y 446.179,Z 493.535,A -85,B 0,C 180,E1 -8555.423,E2 -8555.423} C_VEL
LIN {X 0,Y 446.036,Z 493.832,A -85,B 0,C 180,E1 -8556.94,E2 -8556.94} C_VEL
LIN {X 0,Y 445.904,Z 496.481,A -85,B 0,C 180,E1 -8559.984,E2 -8559.984} C_VEL
LIN {X 0,Y 445.854,Z 498.916,A -85,B 0,C 180,E1 -8562.749,E2 -8562.749} C_VEL
LIN {X 0,Y 445.744,Z 501.713,A -85,B 0,C 180,E1 -8565.89,E2 -8565.89} C_VEL
LIN {X 0,Y 445.72,Z 502.913,A -85,B 0,C 180,E1 -8567.226,E2 -8567.226} C_VEL
LIN {X 0,Y 449.104,Z 513.153,A -85,B 0,C 180,E1 -8567.65,E2 -8567.65} C_VEL
LIN {X 0,Y 453.522,Z 527.487,A -85,B 0,C 180,E1 -8568.347,E2 -8568.347} C_VEL
LIN {X 0,Y 453.801,Z 530.503,A -85,B 0,C 180,E1 -8568.482,E2 -8568.482} C_VEL
LIN {X 0,Y 453.124,Z 544.684,A -85,B 0,C 180,E1 -8569.126,E2 -8569.126} C_VEL
LIN {X 0,Y 452.343,Z 557.533,A -85,B 0,C 180,E1 -8569.869,E2 -8569.869} C_VEL
LIN {X 0,Y 451.354,Z 571.729,A -85,B 0,C 180,E1 -8570.89,E2 -8570.89} C_VEL
LIN {X 0,Y 450.444,Z 584.183,A -85,B 0,C 180,E1 -8571.991,E2 -8571.991} C_VEL
LIN {X 0,Y 449.398,Z 596.143,A -85,B 0,C 180,E1 -8573.258,E2 -8573.258} C_VEL
LIN {X 0,Y 448.521,Z 607.113,A -85,B 0,C 180,E1 -8574.656,E2 -8574.656} C_VEL
LIN {X 0,Y 447.72,Z 616.498,A -85,B 0,C 180,E1 -8576.074,E2 -8576.074} C_VEL
LIN {X 0,Y 447.003,Z 625.172,A -85,B 0,C 180,E1 -8577.633,E2 -8577.633} C_VEL
LIN {X 0,Y 446.492,Z 632.434,A -85,B 0,C 180,E1 -8579.206,E2 -8579.206} C_VEL
LIN {X 0,Y 446.07,Z 638.516,A -85,B 0,C 180,E1 -8580.8,E2 -8580.8} C_VEL
LIN {X 0,Y 445.807,Z 643.531,A -85,B 0,C 180,E1 -8582.412,E2 -8582.412} C_VEL
LIN {X 0,Y 445.589,Z 647.578,A -85,B 0,C 180,E1 -8584.05,E2 -8584.05} C_VEL
LIN {X 0,Y 445.412,Z 650.587,A -85,B 0,C 180,E1 -8585.719,E2 -8585.719} C_VEL
LIN {X 0,Y 445.323,Z 652.09,A -85,B 0,C 180,E1 -8586.849,E2 -8586.849} C_VEL
LIN {X 0,Y 445.292,Z 653.155,A -85,B 0,C 180,E1 -8587.99,E2 -8587.99} C_VEL
LIN {X 0,Y 445.263,Z 653.784,A -85,B 0,C 180,E1 -8589.338,E2 -8589.338} C_VEL
LIN {X 0,Y 445.26,Z 653.808,A -85,B 0,C 180,E1 -8590.743,E2 -8590.743} C_VEL
LIN {X 0,Y 445.321,Z 652.682,A -85,B 0,C 180,E1 -8592.736,E2 -8592.736} C_VEL
LIN {X 0,Y 445.389,Z 651.318,A -85,B 0,C 180,E1 -8593.971,E2 -8593.971} C_VEL
LIN {X 0,Y 445.609,Z 647.739,A -85,B 0,C 180,E1 -8596.055,E2 -8596.055} C_VEL
LIN {X 0,Y 445.921,Z 642.353,A -85,B 0,C 180,E1 -8598.184,E2 -8598.184} C_VEL
LIN {X 0,Y 446.212,Z 637.144,A -85,B 0,C 180,E1 -8599.776,E2 -8599.776} C_VEL
LIN {X 0,Y 446.698,Z 630.331,A -85,B 0,C 180,E1 -8601.457,E2 -8601.457} C_VEL
LIN {X 0,Y 447.287,Z 622.6,A -85,B 0,C 180,E1 -8603.032,E2 -8603.032} C_VEL
LIN {X 0,Y 448.084,Z 613.076,A -85,B 0,C 180,E1 -8604.646,E2 -8604.646} C_VEL
LIN {X 0,Y 449.001,Z 603.101,A -85,B 0,C 180,E1 -8606.055,E2 -8606.055} C_VEL
LIN {X 0,Y 449.975,Z 591.572,A -85,B 0,C 180,E1 -8607.421,E2 -8607.421} C_VEL
LIN {X 0,Y 450.979,Z 579.182,A -85,B 0,C 180,E1 -8608.641,E2 -8608.641} C_VEL
LIN {X 0,Y 451.9,Z 566.956,A -85,B 0,C 180,E1 -8609.639,E2 -8609.639} C_VEL
LIN {X 0,Y 452.757,Z 554.009,A -85,B 0,C 180,E1 -8610.508,E2 -8610.508} C_VEL
LIN {X 0,Y 453.617,Z 539.099,A -85,B 0,C 180,E1 -8611.295,E2 -8611.295} C_VEL
LIN {X 0,Y 453.851,Z 528.361,A -85,B 0,C 180,E1 -8611.753,E2 -8611.753} C_VEL
LIN {X 0,Y 449.418,Z 514.455,A -85,B 0,C 180,E1 -8612.456,E2 -8612.456} C_VEL
LIN {X 0,Y 445.827,Z 504.226,A -85,B 0,C 180,E1 -8612.923,E2 -8612.923} C_VEL
LIN {X 0,Y 445.884,Z 501.612,A -85,B 0,C 180,E1 -8616.09,E2 -8616.09} C_VEL
LIN {X 0,Y 446.006,Z 499.46,A -85,B 0,C 180,E1 -8618.75,E2 -8618.75} C_VEL
LIN {X 0,Y 446.086,Z 497.173,A -85,B 0,C 180,E1 -8621.633,E2 -8621.633} C_VEL
LIN {X 0,Y 446.191,Z 494.929,A -85,B 0,C 180,E1 -8624.468,E2 -8624.468} C_VEL
LIN {X 0,Y 446.24,Z 493.528,A -85,B 0,C 180,E1 -8626.335,E2 -8626.335} C_VEL
LIN {X 0,Y 446.451,Z 493.5,A -85,B 0,C 180,E1 -8629.111,E2 -8629.111} C_VEL
LIN {X 0,Y 446.647,Z 493.475,A -85,B 0,C 180,E1 -8632.435,E2 -8632.435} C_VEL
LIN {X 0,Y 446.645,Z 493.474,A -85,B 0,C 180,E1 -8634.582,E2 -8634.582} C_VEL
LIN {X 0,Y 446.707,Z 493.466,A -85,B 0,C 180,E1 -8637.294,E2 -8637.294} C_VEL
LIN {X 0,Y 446.79,Z 493.457,A -85,B 0,C 180,E1 -8640,E2 -8640} C_VEL
LIN {X 0,Y 446.705,Z 493.465,A -85,B 0,C 180,E1 -8642.705,E2 -8642.705} C_VEL
LIN {X 0,Y 446.645,Z 493.472,A -85,B 0,C 180,E1 -8646.323,E2 -8646.323} C_VEL
LIN {X 0,Y 446.535,Z 493.489,A -85,B 0,C 180,E1 -8649.055,E2 -8649.055} C_VEL
LIN {X 0,Y 446.517,Z 493.492,A -85,B 0,C 180,E1 -8652.73,E2 -8652.73} C_VEL
LIN {X 0,Y 446.492,Z 493.492,A -85,B 0,C 180,E1 -8656.228,E2 -8656.228} C_VEL
LIN {X 0,Y 446.466,Z 493.494,A -85,B 0,C 180,E1 -8659.303,E2 -8659.303} C_VEL
LIN {X 0,Y 446.415,Z 493.504,A -85,B 0,C 180,E1 -8662.199,E2 -8662.199} C_VEL
LIN {X 0,Y 446.455,Z 493.495,A -85,B 0,C 180,E1 -8665.152,E2 -8665.152} C_VEL
LIN {X 0,Y 446.481,Z 493.496,A -85,B 0,C 180,E1 -8668.179,E2 -8668.179} C_VEL
LIN {X 0,Y 446.417,Z 493.504,A -85,B 0,C 180,E1 -8671.3,E2 -8671.3} C_VEL
LIN {X 0,Y 446.427,Z 493.5,A -85,B 0,C 180,E1 -8674.523,E2 -8674.523} C_VEL
LIN {X 0,Y 446.428,Z 493.5,A -85,B 0,C 180,E1 -8678.082,E2 -8678.082} C_VEL
LIN {X 0,Y 446.445,Z 493.5,A -85,B 0,C 180,E1 -8680.921,E2 -8680.921} C_VEL
LIN {X 0,Y 447.192,Z 497.777,A -85,B 0,C 180,E1 -8683.748,E2 -8683.748} C_VEL
LIN {X 0,Y 448.126,Z 503.174,A -85,B 0,C 180,E1 -8686.959,E2 -8686.959} C_VEL
LIN {X 0,Y 448.316,Z 506.633,A -85,B 0,C 180,E1 -8688.822,E2 -8688.822} C_VEL
LIN {X 0,Y 447.873,Z 512.423,A -85,B 0,C 180,E1 -8691.683,E2 -8691.683} C_VEL
LIN {X 0,Y 447.527,Z 519.012,A -85,B 0,C 180,E1 -8694.747,E2 -8694.747} C_VEL
LIN {X 0,Y 447.115,Z 526.624,A -85,B 0,C 180,E1 -8698.081,E2 -8698.081} C_VEL
LIN {X 0,Y 446.692,Z 534.414,A -85,B 0,C 180,E1 -8701.324,E2 -8701.324} C_VEL
LIN {X 0,Y 446.424,Z 541.938,A -85,B 0,C 180,E1 -8704.346,E2 -8704.346} C_VEL
LIN {X 0,Y 446.188,Z 548.989,A -85,B 0,C 180,E1 -8707.1,E2 -8707.1} C_VEL
LIN {X 0,Y 450.097,Z 565.971,A -85,B 0,C 180,E1 -8707.697,E2 -8707.697} C_VEL
LIN {X 0,Y 452.926,Z 580.829,A -85,B 0,C 180,E1 -8708.357,E2 -8708.357} C_VEL
LIN {X 0,Y 453.252,Z 582.396,A -85,B 0,C 180,E1 -8708.435,E2 -8708.435} C_VEL
LIN {X 0,Y 452.477,Z 597.378,A -85,B 0,C 180,E1 -8709.129,E2 -8709.129} C_VEL
LIN {X 0,Y 451.448,Z 611.607,A -85,B 0,C 180,E1 -8709.971,E2 -8709.971} C_VEL
LIN {X 0,Y 450.403,Z 625.372,A -85,B 0,C 180,E1 -8710.99,E2 -8710.99} C_VEL
LIN {X 0,Y 449.43,Z 637.987,A -85,B 0,C 180,E1 -8712.128,E2 -8712.128} C_VEL
LIN {X 0,Y 448.542,Z 649.799,A -85,B 0,C 180,E1 -8713.404,E2 -8713.404} C_VEL
LIN {X 0,Y 447.666,Z 660.358,A -85,B 0,C 180,E1 -8714.754,E2 -8714.754} C_VEL
LIN {X 0,Y 446.917,Z 670.858,A -85,B 0,C 180,E1 -8716.356,E2 -8716.356} C_VEL
LIN {X 0,Y 446.397,Z 678.801,A -85,B 0,C 180,E1 -8717.798,E2 -8717.798} C_VEL
LIN {X 0,Y 445.955,Z 686.887,A -85,B 0,C 180,E1 -8719.558,E2 -8719.558} C_VEL
LIN {X 0,Y 445.665,Z 693.653,A -85,B 0,C 180,E1 -8721.384,E2 -8721.384} C_VEL
LIN {X 0,Y 445.498,Z 698.955,A -85,B 0,C 180,E1 -8723.205,E2 -8723.205} C_VEL
LIN {X 0,Y 445.454,Z 702.027,A -85,B 0,C 180,E1 -8724.568,E2 -8724.568} C_VEL
LIN {X 0,Y 445.431,Z 705.029,A -85,B 0,C 180,E1 -8726.381,E2 -8726.381} C_VEL
LIN {X 0,Y 445.435,Z 706.83,A -85,B 0,C 180,E1 -8728.191,E2 -8728.191} C_VEL
LIN {X 0,Y 445.396,Z 707.46,A -85,B 0,C 180,E1 -8730,E2 -8730} C_VEL
LIN {X 0,Y 445.434,Z 706.875,A -85,B 0,C 180,E1 -8731.808,E2 -8731.808} C_VEL
LIN {X 0,Y 445.416,Z 705.119,A -85,B 0,C 180,E1 -8733.618,E2 -8733.618} C_VEL
LIN {X 0,Y 445.456,Z 702.17,A -85,B 0,C 180,E1 -8735.431,E2 -8735.431} C_VEL
LIN {X 0,Y 445.57,Z 697.959,A -85,B 0,C 180,E1 -8737.249,E2 -8737.249} C_VEL
LIN {X 0,Y 445.72,Z 692.373,A -85,B 0,C 180,E1 -8739.071,E2 -8739.071} C_VEL
LIN {X 0,Y 446.111,Z 685.273,A -85,B 0,C 180,E1 -8740.897,E2 -8740.897} C_VEL
LIN {X 0,Y 446.504,Z 677.081,A -85,B 0,C 180,E1 -8742.61,E2 -8742.61} C_VEL
LIN {X 0,Y 447.153,Z 668.535,A -85,B 0,C 180,E1 -8744.099,E2 -8744.099} C_VEL
LIN {X 0,Y 447.952,Z 657.532,A -85,B 0,C 180,E1 -8745.701,E2 -8745.701} C_VEL
LIN {X 0,Y 448.901,Z 645.712,A -85,B 0,C 180,E1 -8747.128,E2 -8747.128} C_VEL
LIN {X 0,Y 449.842,Z 633.857,A -85,B 0,C 180,E1 -8748.325,E2 -8748.325} C_VEL
LIN {X 0,Y 450.953,Z 620.253,A -85,B 0,C 180,E1 -8749.458,E2 -8749.458} C_VEL
LIN {X 0,Y 451.902,Z 606.916,A -85,B 0,C 180,E1 -8750.363,E2 -8750.363} C_VEL
LIN {X 0,Y 452.816,Z 592.433,A -85,B 0,C 180,E1 -8751.147,E2 -8751.147} C_VEL
LIN {X 0,Y 453.217,Z 581.858,A -85,B 0,C 180,E1 -8751.605,E2 -8751.605} C_VEL
LIN {X 0,Y 450.087,Z 566.668,A -85,B 0,C 180,E1 -8752.284,E2 -8752.284} C_VEL
LIN {X 0,Y 446.255,Z 550.071,A -85,B 0,C 180,E1 -8752.878,E2 -8752.878} C_VEL
LIN {X 0,Y 446.542,Z 543.091,A -85,B 0,C 180,E1 -8755.645,E2 -8755.645} C_VEL
LIN {X 0,Y 446.848,Z 535.644,A -85,B 0,C 180,E1 -8758.67,E2 -8758.67} C_VEL
LIN {X 0,Y 447.148,Z 529.469,A -85,B 0,C 180,E1 -8761.242,E2 -8761.242} C_VEL
LIN {X 0,Y 447.566,Z 522.089,A -85,B 0,C 180,E1 -8764.422,E2 -8764.422} C_VEL
LIN {X 0,Y 447.985,Z 514.724,A -85,B 0,C 180,E1 -8767.721,E2 -8767.721} C_VEL
LIN {X 0,Y 448.44,Z 508.643,A -85,B 0,C 180,E1 -8770.57,E2 -8770.57} C_VEL
LIN {X 0,Y 448.39,Z 504.632,A -85,B 0,C 180,E1 -8772.552,E2 -8772.552} C_VEL
LIN {X 0,Y 447.622,Z 499.932,A -85,B 0,C 180,E1 -8775.047,E2 -8775.047} C_VEL
LIN {X 0,Y 446.761,Z 495.245,A -85,B 0,C 180,E1 -8777.675,E2 -8777.675} C_VEL
LIN {X 0,Y 446.464,Z 493.499,A -85,B 0,C 180,E1 -8778.748,E2 -8778.748} C_VEL
LIN {X 0,Y 446.47,Z 493.499,A -85,B 0,C 180,E1 -8780.976,E2 -8780.976} C_VEL
LIN {X 0,Y 446.413,Z 493.504,A -85,B 0,C 180,E1 -8784.374,E2 -8784.374} C_VEL
LIN {X 0,Y 446.414,Z 493.505,A -85,B 0,C 180,E1 -8787.638,E2 -8787.638} C_VEL
LIN {X 0,Y 446.46,Z 493.497,A -85,B 0,C 180,E1 -8790.792,E2 -8790.792} C_VEL
LIN {X 0,Y 446.468,Z 493.499,A -85,B 0,C 180,E1 -8793.848,E2 -8793.848} C_VEL
LIN {X 0,Y 446.419,Z 493.502,A -85,B 0,C 180,E1 -8796.823,E2 -8796.823} C_VEL
LIN {X 0,Y 446.434,Z 493.502,A -85,B 0,C 180,E1 -8799.737,E2 -8799.737} C_VEL
LIN {X 0,Y 446.455,Z 493.496,A -85,B 0,C 180,E1 -8802.597,E2 -8802.597} C_VEL
LIN {X 0,Y 446.463,Z 493.5,A -85,B 0,C 180,E1 -8805.412,E2 -8805.412} C_VEL
LIN {X 0,Y 446.53,Z 493.489,A -85,B 0,C 180,E1 -8808.194,E2 -8808.194} C_VEL
LIN {X 0,Y 446.59,Z 493.482,A -85,B 0,C 180,E1 -8811.858,E2 -8811.858} C_VEL
LIN {X 0,Y 446.64,Z 493.473,A -85,B 0,C 180,E1 -8814.583,E2 -8814.583} C_VEL
LIN {X 0,Y 446.702,Z 493.469,A -85,B 0,C 180,E1 -8817.295,E2 -8817.295} C_VEL
LIN {X 0,Y 446.784,Z 493.458,A -85,B 0,C 180,E1 -8820,E2 -8820} C_VEL
LIN {X 0,Y 446.702,Z 493.466,A -85,B 0,C 180,E1 -8822.706,E2 -8822.706} C_VEL
LIN {X 0,Y 446.643,Z 493.473,A -85,B 0,C 180,E1 -8826.324,E2 -8826.324} C_VEL
LIN {X 0,Y 446.529,Z 493.489,A -85,B 0,C 180,E1 -8829.056,E2 -8829.056} C_VEL
LIN {X 0,Y 446.512,Z 493.49,A -85,B 0,C 180,E1 -8832.73,E2 -8832.73} C_VEL
LIN {X 0,Y 446.487,Z 493.493,A -85,B 0,C 180,E1 -8836.229,E2 -8836.229} C_VEL
LIN {X 0,Y 446.461,Z 493.499,A -85,B 0,C 180,E1 -8839.304,E2 -8839.304} C_VEL
LIN {X 0,Y 446.41,Z 493.504,A -85,B 0,C 180,E1 -8842.2,E2 -8842.2} C_VEL
LIN {X 0,Y 446.451,Z 493.5,A -85,B 0,C 180,E1 -8845.153,E2 -8845.153} C_VEL
LIN {X 0,Y 446.477,Z 493.495,A -85,B 0,C 180,E1 -8848.18,E2 -8848.18} C_VEL
LIN {X 0,Y 446.424,Z 493.503,A -85,B 0,C 180,E1 -8851.3,E2 -8851.3} C_VEL
LIN {X 0,Y 446.425,Z 493.501,A -85,B 0,C 180,E1 -8854.524,E2 -8854.524} C_VEL
LIN {X 0,Y 446.435,Z 493.5,A -85,B 0,C 180,E1 -8858.084,E2 -8858.084} C_VEL
LIN {X 0,Y 446.444,Z 493.499,A -85,B 0,C 180,E1 -8860.922,E2 -8860.922} C_VEL
LIN {X 0,Y 446.442,Z 493.501,A -85,B 0,C 180,E1 -8863.842,E2 -8863.842} C_VEL
LIN {X 0,Y 446.444,Z 493.498,A -85,B 0,C 180,E1 -8866.398,E2 -8866.398} C_VEL
LIN {X 0,Y 446.467,Z 493.499,A -85,B 0,C 180,E1 -8869.806,E2 -8869.806} C_VEL
LIN {X 0,Y 446.433,Z 493.501,A -85,B 0,C 180,E1 -8872.125,E2 -8872.125} C_VEL
LIN {X 0,Y 446.43,Z 493.503,A -85,B 0,C 180,E1 -8875.478,E2 -8875.478} C_VEL
LIN {X 0,Y 446.417,Z 493.501,A -85,B 0,C 180,E1 -8878.701,E2 -8878.701} C_VEL
LIN {X 0,Y 446.485,Z 493.496,A -85,B 0,C 180,E1 -8881.823,E2 -8881.823} C_VEL
LIN {X 0,Y 446.46,Z 493.497,A -85,B 0,C 180,E1 -8884.849,E2 -8884.849} C_VEL
LIN {X 0,Y 446.451,Z 493.498,A -85,B 0,C 180,E1 -8888.246,E2 -8888.246} C_VEL
LIN {X 0,Y 446.461,Z 493.499,A -85,B 0,C 180,E1 -8891.65,E2 -8891.65} C_VEL
LIN {X 0,Y 446.512,Z 493.49,A -85,B 0,C 180,E1 -8894.481,E2 -8894.481} C_VEL
LIN {X 0,Y 446.521,Z 493.49,A -85,B 0,C 180,E1 -8898.194,E2 -8898.194} C_VEL
LIN {X 0,Y 446.537,Z 493.487,A -85,B 0,C 180,E1 -8900.945,E2 -8900.945} C_VEL
LIN {X 0,Y 446.646,Z 493.476,A -85,B 0,C 180,E1 -8903.677,E2 -8903.677} C_VEL
LIN {X 0,Y 446.631,Z 493.475,A -85,B 0,C 180,E1 -8907.015,E2 -8907.015} C_VEL
LIN {X 0,Y 446.115,Z 493.543,A -85,B 0,C 180,E1 -8907.768,E2 -8907.768} C_VEL
LIN {X 0,Y 443.301,Z 493.894,A -85,B 0,C 180,E1 -8908.991,E2 -8908.991} C_VEL
LIN {X 0,Y 440.808,Z 494.203,A -85,B 0,C 180,E1 -8909.977,E2 -8909.977} C_VEL
LIN {X 0,Y 439.706,Z 494.338,A -85,B 0,C 180,E1 -8910.741,E2 -8910.741} C_VEL
LIN {X 0,Y 439.605,Z 494.35,A -85,B 0,C 180,E1 -8911,E2 -8911} C_VEL
LIN {X 0,Y 439.442,Z 494.371,A -85,B 0,C 180,E1 -8912.75,E2 -8912.75} C_VEL
LIN {X 0,Y 439.126,Z 494.414,A -85,B 0,C 180,E1 -8915.511,E2 -8915.511} C_VEL
LIN {X 0,Y 438.984,Z 494.629,A -85,B 0,C 180,E1 -8916.969,E2 -8916.969} C_VEL
LIN {X 0,Y 438.833,Z 497.38,A -85,B 0,C 180,E1 -8920.147,E2 -8920.147} C_VEL
LIN {X 0,Y 438.766,Z 499.821,A -85,B 0,C 180,E1 -8922.959,E2 -8922.959} C_VEL
LIN {X 0,Y 438.681,Z 502.533,A -85,B 0,C 180,E1 -8926.001,E2 -8926.001} C_VEL
LIN {X 0,Y 438.668,Z 503.279,A -85,B 0,C 180,E1 -8926.842,E2 -8926.842} C_VEL
LIN {X 0,Y 441.195,Z 510.919,A -85,B 0,C 180,E1 -8927.164,E2 -8927.164} C_VEL
LIN {X 0,Y 445.873,Z 525.267,A -85,B 0,C 180,E1 -8927.862,E2 -8927.862} C_VEL
LIN {X 0,Y 447.213,Z 530.428,A -85,B 0,C 180,E1 -8928.14,E2 -8928.14} C_VEL
LIN {X 0,Y 446.521,Z 544.193,A -85,B 0,C 180,E1 -8928.765,E2 -8928.765} C_VEL
LIN {X 0,Y 445.647,Z 558.178,A -85,B 0,C 180,E1 -8929.58,E2 -8929.58} C_VEL
LIN {X 0,Y 444.62,Z 572.544,A -85,B 0,C 180,E1 -8930.634,E2 -8930.634} C_VEL
LIN {X 0,Y 443.667,Z 584.762,A -85,B 0,C 180,E1 -8931.733,E2 -8931.733} C_VEL
LIN {X 0,Y 442.627,Z 596.025,A -85,B 0,C 180,E1 -8932.938,E2 -8932.938} C_VEL
LIN {X 0,Y 441.757,Z 605.89,A -85,B 0,C 180,E1 -8934.184,E2 -8934.184} C_VEL
LIN {X 0,Y 440.85,Z 616.274,A -85,B 0,C 180,E1 -8935.748,E2 -8935.748} C_VEL
LIN {X 0,Y 440.125,Z 625.043,A -85,B 0,C 180,E1 -8937.334,E2 -8937.334} C_VEL
LIN {X 0,Y 439.474,Z 633.489,A -85,B 0,C 180,E1 -8939.193,E2 -8939.193} C_VEL
LIN {X 0,Y 439.021,Z 639.474,A -85,B 0,C 180,E1 -8940.815,E2 -8940.815} C_VEL
LIN {X 0,Y 438.743,Z 644.369,A -85,B 0,C 180,E1 -8942.453,E2 -8942.453} C_VEL
LIN {X 0,Y 438.497,Z 648.314,A -85,B 0,C 180,E1 -8944.122,E2 -8944.122} C_VEL
LIN {X 0,Y 438.396,Z 650.369,A -85,B 0,C 180,E1 -8945.248,E2 -8945.248} C_VEL
LIN {X 0,Y 438.247,Z 652.38,A -85,B 0,C 180,E1 -8946.694,E2 -8946.694} C_VEL
LIN {X 0,Y 438.179,Z 653.994,A -85,B 0,C 180,E1 -8948.72,E2 -8948.72} C_VEL
LIN {X 0,Y 438.169,Z 654.321,A -85,B 0,C 180,E1 -8949.909,E2 -8949.909} C_VEL
LIN {X 0,Y 438.18,Z 654.167,A -85,B 0,C 180,E1 -8951.117,E2 -8951.117} C_VEL
LIN {X 0,Y 438.227,Z 653.379,A -85,B 0,C 180,E1 -8952.462,E2 -8952.462} C_VEL
LIN {X 0,Y 438.295,Z 652.011,A -85,B 0,C 180,E1 -8953.815,E2 -8953.815} C_VEL
LIN {X 0,Y 438.434,Z 650.082,A -85,B 0,C 180,E1 -8955.145,E2 -8955.145} C_VEL
LIN {X 0,Y 438.646,Z 646.295,A -85,B 0,C 180,E1 -8956.991,E2 -8956.991} C_VEL
LIN {X 0,Y 438.963,Z 640.826,A -85,B 0,C 180,E1 -8958.971,E2 -8958.971} C_VEL
LIN {X 0,Y 439.477,Z 634.203,A -85,B 0,C 180,E1 -8960.826,E2 -8960.826} C_VEL
LIN {X 0,Y 440.11,Z 626.149,A -85,B 0,C 180,E1 -8962.64,E2 -8962.64} C_VEL
LIN {X 0,Y 440.977,Z 616.724,A -85,B 0,C 180,E1 -8964.37,E2 -8964.37} C_VEL
LIN {X 0,Y 441.937,Z 605.955,A -85,B 0,C 180,E1 -8965.997,E2 -8965.997} C_VEL
LIN {X 0,Y 442.947,Z 595.159,A -85,B 0,C 180,E1 -8967.353,E2 -8967.353} C_VEL
LIN {X 0,Y 443.985,Z 583.186,A -85,B 0,C 180,E1 -8968.61,E2 -8968.61} C_VEL
LIN {X 0,Y 445.003,Z 570.41,A -85,B 0,C 180,E1 -8969.721,E2 -8969.721} C_VEL
LIN {X 0,Y 445.94,Z 557.18,A -85,B 0,C 180,E1 -8970.661,E2 -8970.661} C_VEL
LIN {X 0,Y 446.878,Z 543.08,A -85,B 0,C 180,E1 -8971.456,E2 -8971.456} C_VEL
LIN {X 0,Y 447.339,Z 530.086,A -85,B 0,C 180,E1 -8972.039,E2 -8972.039} C_VEL
LIN {X 0,Y 442.756,Z 515.893,A -85,B 0,C 180,E1 -8972.797,E2 -8972.797} C_VEL
LIN {X 0,Y 438.816,Z 504.951,A -85,B 0,C 180,E1 -8973.298,E2 -8973.298} C_VEL
LIN {X 0,Y 438.782,Z 504.362,A -85,B 0,C 180,E1 -8973.76,E2 -8973.76} C_VEL
LIN {X 0,Y 438.851,Z 502.229,A -85,B 0,C 180,E1 -8976.399,E2 -8976.399} C_VEL
LIN {X 0,Y 438.949,Z 499.84,A -85,B 0,C 180,E1 -8979.375,E2 -8979.375} C_VEL
LIN {X 0,Y 439.06,Z 497.551,A -85,B 0,C 180,E1 -8982.294,E2 -8982.294} C_VEL
LIN {X 0,Y 439.155,Z 495.334,A -85,B 0,C 180,E1 -8985.163,E2 -8985.163} C_VEL
LIN {X 0,Y 439.181,Z 494.611,A -85,B 0,C 180,E1 -8986.111,E2 -8986.111} C_VEL
LIN {X 0,Y 439.4,Z 494.383,A -85,B 0,C 180,E1 -8987.999,E2 -8987.999} C_VEL
LIN {X 0,Y 439.495,Z 494.365,A -85,B 0,C 180,E1 -8990.798,E2 -8990.798} C_VEL
LIN {X 0,Y 439.616,Z 494.351,A -85,B 0,C 180,E1 -8993.574,E2 -8993.574} C_VEL
LIN {X 0,Y 439.654,Z 494.344,A -85,B 0,C 180,E1 -8997.251,E2 -8997.251} C_VEL
LIN {X 0,Y 439.76,Z 494.333,A -85,B 0,C 180,E1 -9000,E2 -9000} C_VEL
LIN {X 0,Y 439.652,Z 494.344,A -85,B 0,C 180,E1 -9002.748,E2 -9002.748} C_VEL
LIN {X 0,Y 439.616,Z 494.348,A -85,B 0,C 180,E1 -9006.425,E2 -9006.425} C_VEL
LIN {X 0,Y 439.497,Z 494.365,A -85,B 0,C 180,E1 -9009.201,E2 -9009.201} C_VEL
LIN {X 0,Y 439.462,Z 494.369,A -85,B 0,C 180,E1 -9012.937,E2 -9012.937} C_VEL
LIN {X 0,Y 439.443,Z 494.371,A -85,B 0,C 180,E1 -9016.349,E2 -9016.349} C_VEL
LIN {X 0,Y 439.399,Z 494.373,A -85,B 0,C 180,E1 -9019.626,E2 -9019.626} C_VEL
LIN {X 0,Y 439.362,Z 494.382,A -85,B 0,C 180,E1 -9022.575,E2 -9022.575} C_VEL
LIN {X 0,Y 439.402,Z 494.375,A -85,B 0,C 180,E1 -9025.585,E2 -9025.585} C_VEL
LIN {X 0,Y 439.422,Z 494.375,A -85,B 0,C 180,E1 -9028.673,E2 -9028.673} C_VEL
LIN {X 0,Y 439.371,Z 494.382,A -85,B 0,C 180,E1 -9031.86,E2 -9031.86} C_VEL
LIN {X 0,Y 439.398,Z 494.378,A -85,B 0,C 180,E1 -9035.156,E2 -9035.156} C_VEL
LIN {X 0,Y 439.381,Z 494.373,A -85,B 0,C 180,E1 -9038.595,E2 -9038.595} C_VEL
LIN {X 0,Y 439.437,Z 494.457,A -85,B 0,C 180,E1 -9040.52,E2 -9040.52} C_VEL
LIN {X 0,Y 440.314,Z 499.765,A -85,B 0,C 180,E1 -9044.089,E2 -9044.089} C_VEL
LIN {X 0,Y 441.218,Z 504.797,A -85,B 0,C 180,E1 -9047.114,E2 -9047.114} C_VEL
LIN {X 0,Y 441.274,Z 508.732,A -85,B 0,C 180,E1 -9049.233,E2 -9049.233} C_VEL
LIN {X 0,Y 440.818,Z 514.57,A -85,B 0,C 180,E1 -9052.135,E2 -9052.135} C_VEL
LIN {X 0,Y 440.456,Z 520.536,A -85,B 0,C 180,E1 -9054.941,E2 -9054.941} C_VEL
LIN {X 0,Y 440.054,Z 527.86,A -85,B 0,C 180,E1 -9058.195,E2 -9058.195} C_VEL
LIN {X 0,Y 439.633,Z 535.756,A -85,B 0,C 180,E1 -9061.55,E2 -9061.55} C_VEL
LIN {X 0,Y 439.336,Z 542.757,A -85,B 0,C 180,E1 -9064.411,E2 -9064.411} C_VEL
LIN {X 0,Y 439.124,Z 548.495,A -85,B 0,C 180,E1 -9066.695,E2 -9066.695} C_VEL
LIN {X 0,Y 443.147,Z 565.473,A -85,B 0,C 180,E1 -9067.32,E2 -9067.32} C_VEL
LIN {X 0,Y 446.111,Z 581.461,A -85,B 0,C 180,E1 -9068.05,E2 -9068.05} C_VEL
LIN {X 0,Y 446.479,Z 585.194,A -85,B 0,C 180,E1 -9068.235,E2 -9068.235} C_VEL
LIN {X 0,Y 445.616,Z 600.038,A -85,B 0,C 180,E1 -9068.973,E2 -9068.973} C_VEL
LIN {X 0,Y 444.616,Z 612.862,A -85,B 0,C 180,E1 -9069.771,E2 -9069.771} C_VEL
LIN {X 0,Y 443.51,Z 626.32,A -85,B 0,C 180,E1 -9070.803,E2 -9070.803} C_VEL
LIN {X 0,Y 442.434,Z 639.82,A -85,B 0,C 180,E1 -9072.075,E2 -9072.075} C_VEL
LIN {X 0,Y 441.519,Z 651.138,A -85,B 0,C 180,E1 -9073.35,E2 -9073.35} C_VEL
LIN {X 0,Y 440.597,Z 661.546,A -85,B 0,C 180,E1 -9074.74,E2 -9074.74} C_VEL
LIN {X 0,Y 439.812,Z 671.768,A -85,B 0,C 180,E1 -9076.367,E2 -9076.367} C_VEL
LIN {X 0,Y 439.284,Z 680.283,A -85,B 0,C 180,E1 -9077.996,E2 -9077.996} C_VEL
LIN {X 0,Y 438.924,Z 686.43,A -85,B 0,C 180,E1 -9079.389,E2 -9079.389} C_VEL
LIN {X 0,Y 438.577,Z 693.201,A -85,B 0,C 180,E1 -9081.243,E2 -9081.243} C_VEL
LIN {X 0,Y 438.434,Z 698.513,A -85,B 0,C 180,E1 -9083.095,E2 -9083.095} C_VEL
LIN {X 0,Y 438.374,Z 701.588,A -85,B 0,C 180,E1 -9084.48,E2 -9084.48} C_VEL
LIN {X 0,Y 438.332,Z 704.595,A -85,B 0,C 180,E1 -9086.322,E2 -9086.322} C_VEL
LIN {X 0,Y 438.35,Z 706.4,A -85,B 0,C 180,E1 -9088.162,E2 -9088.162} C_VEL
LIN {X 0,Y 438.334,Z 707.035,A -85,B 0,C 180,E1 -9090,E2 -9090} C_VEL
LIN {X 0,Y 438.35,Z 706.45,A -85,B 0,C 180,E1 -9091.837,E2 -9091.837} C_VEL
LIN {X 0,Y 438.318,Z 704.692,A -85,B 0,C 180,E1 -9093.677,E2 -9093.677} C_VEL
LIN {X 0,Y 438.38,Z 701.742,A -85,B 0,C 180,E1 -9095.519,E2 -9095.519} C_VEL
LIN {X 0,Y 438.487,Z 697.528,A -85,B 0,C 180,E1 -9097.366,E2 -9097.366} C_VEL
LIN {X 0,Y 438.645,Z 691.937,A -85,B 0,C 180,E1 -9099.219,E2 -9099.219} C_VEL
LIN {X 0,Y 439.09,Z 684.834,A -85,B 0,C 180,E1 -9101.073,E2 -9101.073} C_VEL
LIN {X 0,Y 439.455,Z 677.251,A -85,B 0,C 180,E1 -9102.698,E2 -9102.698} C_VEL
LIN {X 0,Y 440.192,Z 668.086,A -85,B 0,C 180,E1 -9104.327,E2 -9104.327} C_VEL
LIN {X 0,Y 441.051,Z 657.074,A -85,B 0,C 180,E1 -9105.954,E2 -9105.954} C_VEL
LIN {X 0,Y 441.969,Z 646.114,A -85,B 0,C 180,E1 -9107.305,E2 -9107.305} C_VEL
LIN {X 0,Y 443.042,Z 633.385,A -85,B 0,C 180,E1 -9108.616,E2 -9108.616} C_VEL
LIN {X 0,Y 444.18,Z 619.767,A -85,B 0,C 180,E1 -9109.767,E2 -9109.767} C_VEL
LIN {X 0,Y 445.188,Z 606.425,A -85,B 0,C 180,E1 -9110.684,E2 -9110.684} C_VEL
LIN {X 0,Y 446.147,Z 591.917,A -85,B 0,C 180,E1 -9111.478,E2 -9111.478} C_VEL
LIN {X 0,Y 446.618,Z 583.825,A -85,B 0,C 180,E1 -9111.839,E2 -9111.839} C_VEL
LIN {X 0,Y 443.426,Z 567.766,A -85,B 0,C 180,E1 -9112.586,E2 -9112.586} C_VEL
LIN {X 0,Y 439.648,Z 552.016,A -85,B 0,C 180,E1 -9113.162,E2 -9113.162} C_VEL
LIN {X 0,Y 439.209,Z 549.786,A -85,B 0,C 180,E1 -9113.23,E2 -9113.23} C_VEL
LIN {X 0,Y 439.562,Z 541.828,A -85,B 0,C 180,E1 -9116.445,E2 -9116.445} C_VEL
LIN {X 0,Y 439.937,Z 534.052,A -85,B 0,C 180,E1 -9119.683,E2 -9119.683} C_VEL
LIN {X 0,Y 440.419,Z 525.452,A -85,B 0,C 180,E1 -9123.396,E2 -9123.396} C_VEL
LIN {X 0,Y 440.804,Z 518.22,A -85,B 0,C 180,E1 -9126.653,E2 -9126.653} C_VEL
LIN {X 0,Y 441.279,Z 511.982,A -85,B 0,C 180,E1 -9129.571,E2 -9129.571} C_VEL
LIN {X 0,Y 441.496,Z 507.127,A -85,B 0,C 180,E1 -9131.956,E2 -9131.956} C_VEL
LIN {X 0,Y 440.84,Z 502.246,A -85,B 0,C 180,E1 -9134.543,E2 -9134.543} C_VEL
LIN {X 0,Y 439.779,Z 496.438,A -85,B 0,C 180,E1 -9137.841,E2 -9137.841} C_VEL
LIN {X 0,Y 439.427,Z 494.375,A -85,B 0,C 180,E1 -9139.176,E2 -9139.176} C_VEL
LIN {X 0,Y 439.386,Z 494.38,A -85,B 0,C 180,E1 -9141.604,E2 -9141.604} C_VEL
LIN {X 0,Y 439.392,Z 494.377,A -85,B 0,C 180,E1 -9144.844,E2 -9144.844} C_VEL
LIN {X 0,Y 439.365,Z 494.381,A -85,B 0,C 180,E1 -9148.139,E2 -9148.139} C_VEL
LIN {X 0,Y 439.416,Z 494.377,A -85,B 0,C 180,E1 -9151.327,E2 -9151.327} C_VEL
LIN {X 0,Y 439.395,Z 494.376,A -85,B 0,C 180,E1 -9154.415,E2 -9154.415} C_VEL
LIN {X 0,Y 439.355,Z 494.385,A -85,B 0,C 180,E1 -9157.424,E2 -9157.424} C_VEL
LIN {X 0,Y 439.431,Z 494.372,A -85,B 0,C 180,E1 -9160.663,E2 -9160.663} C_VEL
LIN {X 0,Y 439.465,Z 494.367,A -85,B 0,C 180,E1 -9164.225,E2 -9164.225} C_VEL
LIN {X 0,Y 439.498,Z 494.366,A -85,B 0,C 180,E1 -9168.002,E2 -9168.002} C_VEL
LIN {X 0,Y 439.538,Z 494.362,A -85,B 0,C 180,E1 -9171.726,E2 -9171.726} C_VEL
LIN {X 0,Y 439.615,Z 494.348,A -85,B 0,C 180,E1 -9174.496,E2 -9174.496} C_VEL
LIN {X 0,Y 439.626,Z 494.348,A -85,B 0,C 180,E1 -9178.168,E2 -9178.168} C_VEL
LIN {X 0,Y 439.755,Z 494.334,A -85,B 0,C 180,E1 -9180,E2 -9180} C_VEL
LIN {X 0,Y 439.649,Z 494.345,A -85,B 0,C 180,E1 -9182.749,E2 -9182.749} C_VEL
LIN {X 0,Y 439.613,Z 494.348,A -85,B 0,C 180,E1 -9186.426,E2 -9186.426} C_VEL
LIN {X 0,Y 439.491,Z 494.366,A -85,B 0,C 180,E1 -9189.202,E2 -9189.202} C_VEL
LIN {X 0,Y 439.456,Z 494.37,A -85,B 0,C 180,E1 -9192.938,E2 -9192.938} C_VEL
LIN {X 0,Y 439.438,Z 494.37,A -85,B 0,C 180,E1 -9196.35,E2 -9196.35} C_VEL
LIN {X 0,Y 439.394,Z 494.38,A -85,B 0,C 180,E1 -9199.627,E2 -9199.627} C_VEL
LIN {X 0,Y 439.357,Z 494.381,A -85,B 0,C 180,E1 -9202.576,E2 -9202.576} C_VEL
LIN {X 0,Y 439.398,Z 494.379,A -85,B 0,C 180,E1 -9205.586,E2 -9205.586} C_VEL
LIN {X 0,Y 439.418,Z 494.373,A -85,B 0,C 180,E1 -9208.674,E2 -9208.674} C_VEL
LIN {X 0,Y 439.377,Z 494.381,A -85,B 0,C 180,E1 -9212.034,E2 -9212.034} C_VEL
LIN {X 0,Y 439.391,Z 494.38,A -85,B 0,C 180,E1 -9215.342,E2 -9215.342} C_VEL
LIN {X 0,Y 439.396,Z 494.375,A -85,B 0,C 180,E1 -9218.594,E2 -9218.594} C_VEL
LIN {X 0,Y 439.401,Z 494.378,A -85,B 0,C 180,E1 -9221.261,E2 -9221.261} C_VEL
LIN {X 0,Y 439.407,Z 494.375,A -85,B 0,C 180,E1 -9224.729,E2 -9224.729} C_VEL
LIN {X 0,Y 439.41,Z 494.378,A -85,B 0,C 180,E1 -9227.799,E2 -9227.799} C_VEL
LIN {X 0,Y 439.45,Z 494.37,A -85,B 0,C 180,E1 -9230.231,E2 -9230.231} C_VEL
LIN {X 0,Y 439.376,Z 494.382,A -85,B 0,C 180,E1 -9233.714,E2 -9233.714} C_VEL
LIN {X 0,Y 439.372,Z 494.381,A -85,B 0,C 180,E1 -9237.055,E2 -9237.055} C_VEL
LIN {X 0,Y 439.383,Z 494.377,A -85,B 0,C 180,E1 -9240.275,E2 -9240.275} C_VEL
LIN {X 0,Y 439.432,Z 494.375,A -85,B 0,C 180,E1 -9243.398,E2 -9243.398} C_VEL
LIN {X 0,Y 439.389,Z 494.377,A -85,B 0,C 180,E1 -9246.431,E2 -9246.431} C_VEL
LIN {X 0,Y 439.391,Z 494.38,A -85,B 0,C 180,E1 -9249.398,E2 -9249.398} C_VEL
LIN {X 0,Y 439.435,Z 494.371,A -85,B 0,C 180,E1 -9252.311,E2 -9252.311} C_VEL
LIN {X 0,Y 439.452,Z 494.371,A -85,B 0,C 180,E1 -9255.175,E2 -9255.175} C_VEL
LIN {X 0,Y 439.488,Z 494.367,A -85,B 0,C 180,E1 -9258.002,E2 -9258.002} C_VEL
LIN {X 0,Y 439.508,Z 494.366,A -85,B 0,C 180,E1 -9261.726,E2 -9261.726} C_VEL
LIN {X 0,Y 439.625,Z 494.347,A -85,B 0,C 180,E1 -9264.496,E2 -9264.496} C_VEL
LIN {X 0,Y 439.642,Z 494.347,A -85,B 0,C 180,E1 -9268.168,E2 -9268.168} C_VEL
LIN {X 0,Y 439.768,Z 494.332,A -85,B 0,C 180,E1 -9270,E2 -9270} C_VEL
LIN {X 0,Y 439.605,Z 494.35,A -85,B 0,C 180,E1 -9271,E2 -9271} C_VEL
LIN {X 0,Y 438.882,Z 494.444,A -85,B 0,C 180,E1 -9271.762,E2 -9271.762} C_VEL
LIN {X 0,Y 435.896,Z 494.813,A -85,B 0,C 180,E1 -9272.998,E2 -9272.998} C_VEL
LIN {X 0,Y 433.358,Z 495.132,A -85,B 0,C 180,E1 -9273.995,E2 -9273.995} C_VEL
LIN {X 0,Y 432.231,Z 495.27,A -85,B 0,C 180,E1 -9274.768,E2 -9274.768} C_VEL
LIN {X 0,Y 432.119,Z 495.283,A -85,B 0,C 180,E1 -9275.03,E2 -9275.03} C_VEL
LIN {X 0,Y 431.931,Z 495.454,A -85,B 0,C 180,E1 -9276.999,E2 -9276.999} C_VEL
LIN {X 0,Y 431.765,Z 498.293,A -85,B 0,C 180,E1 -9280.315,E2 -9280.315} C_VEL
LIN {X 0,Y 431.708,Z 500.779,A -85,B 0,C 180,E1 -9283.174,E2 -9283.174} C_VEL
LIN {X 0,Y 431.607,Z 503.696,A -85,B 0,C 180,E1 -9286.465,E2 -9286.465} C_VEL
LIN {X 0,Y 436.71,Z 518.814,A -85,B 0,C 180,E1 -9287.142,E2 -9287.142} C_VEL
LIN {X 0,Y 440.582,Z 531.827,A -85,B 0,C 180,E1 -9287.846,E2 -9287.846} C_VEL
LIN {X 0,Y 439.79,Z 547.188,A -85,B 0,C 180,E1 -9288.579,E2 -9288.579} C_VEL
LIN {X 0,Y 438.804,Z 561.262,A -85,B 0,C 180,E1 -9289.447,E2 -9289.447} C_VEL
LIN {X 0,Y 437.81,Z 574.132,A -85,B 0,C 180,E1 -9290.435,E2 -9290.435} C_VEL
LIN {X 0,Y 436.839,Z 586.168,A -85,B 0,C 180,E1 -9291.554,E2 -9291.554} C_VEL
LIN {X 0,Y 435.729,Z 597.248,A -85,B 0,C 180,E1 -9292.774,E2 -9292.774} C_VEL
LIN {X 0,Y 434.795,Z 607.32,A -85,B 0,C 180,E1 -9294.088,E2 -9294.088} C_VEL
LIN {X 0,Y 433.863,Z 617.566,A -85,B 0,C 180,E1 -9295.682,E2 -9295.682} C_VEL
LIN {X 0,Y 433.098,Z 626.174,A -85,B 0,C 180,E1 -9297.285,E2 -9297.285} C_VEL
LIN {X 0,Y 432.519,Z 633.323,A -85,B 0,C 180,E1 -9298.883,E2 -9298.883} C_VEL
LIN {X 0,Y 431.948,Z 640.564,A -85,B 0,C 180,E1 -9300.87,E2 -9300.87} C_VEL
LIN {X 0,Y 431.679,Z 645.213,A -85,B 0,C 180,E1 -9302.497,E2 -9302.497} C_VEL
LIN {X 0,Y 431.47,Z 648.337,A -85,B 0,C 180,E1 -9303.827,E2 -9303.827} C_VEL
LIN {X 0,Y 431.226,Z 651.937,A -85,B 0,C 180,E1 -9305.924,E2 -9305.924} C_VEL
LIN {X 0,Y 431.154,Z 653.282,A -85,B 0,C 180,E1 -9307.093,E2 -9307.093} C_VEL
LIN {X 0,Y 431.096,Z 654.316,A -85,B 0,C 180,E1 -9308.507,E2 -9308.507} C_VEL
LIN {X 0,Y 431.079,Z 654.761,A -85,B 0,C 180,E1 -9309.981,E2 -9309.981} C_VEL
LIN {X 0,Y 431.101,Z 654.208,A -85,B 0,C 180,E1 -9311.943,E2 -9311.943} C_VEL
LIN {X 0,Y 431.201,Z 653.228,A -85,B 0,C 180,E1 -9313.199,E2 -9313.199} C_VEL
LIN {X 0,Y 431.285,Z 651.647,A -85,B 0,C 180,E1 -9314.483,E2 -9314.483} C_VEL
LIN {X 0,Y 431.504,Z 648.479,A -85,B 0,C 180,E1 -9316.319,E2 -9316.319} C_VEL
LIN {X 0,Y 431.86,Z 643.193,A -85,B 0,C 180,E1 -9318.468,E2 -9318.468} C_VEL
LIN {X 0,Y 432.255,Z 637.461,A -85,B 0,C 180,E1 -9320.26,E2 -9320.26} C_VEL
LIN {X 0,Y 432.803,Z 630.958,A -85,B 0,C 180,E1 -9321.898,E2 -9321.898} C_VEL
LIN {X 0,Y 433.547,Z 622.511,A -85,B 0,C 180,E1 -9323.652,E2 -9323.652} C_VEL
LIN {X 0,Y 434.404,Z 613.337,A -85,B 0,C 180,E1 -9325.229,E2 -9325.229} C_VEL
LIN {X 0,Y 435.468,Z 602.942,A -85,B 0,C 180,E1 -9326.72,E2 -9326.72} C_VEL
LIN {X 0,Y 436.529,Z 591.563,A -85,B 0,C 180,E1 -9328.087,E2 -9328.087} C_VEL
LIN {X 0,Y 437.603,Z 579.319,A -85,B 0,C 180,E1 -9329.313,E2 -9329.313} C_VEL
LIN {X 0,Y 438.702,Z 566.706,A -85,B 0,C 180,E1 -9330.355,E2 -9330.355} C_VEL
LIN {X 0,Y 439.697,Z 552.949,A -85,B 0,C 180,E1 -9331.281,E2 -9331.281} C_VEL
LIN {X 0,Y 440.574,Z 538.25,A -85,B 0,C 180,E1 -9332.057,E2 -9332.057} C_VEL
LIN {X 0,Y 440.71,Z 531.545,A -85,B 0,C 180,E1 -9332.357,E2 -9332.357} C_VEL
LIN {X 0,Y 436.124,Z 517.348,A -85,B 0,C 180,E1 -9333.146,E2 -9333.146} C_VEL
LIN {X 0,Y 431.768,Z 505.459,A -85,B 0,C 180,E1 -9333.716,E2 -9333.716} C_VEL
LIN {X 0,Y 431.741,Z 505.074,A -85,B 0,C 180,E1 -9333.927,E2 -9333.927} C_VEL
LIN {X 0,Y 431.808,Z 502.602,A -85,B 0,C 180,E1 -9337.007,E2 -9337.007} C_VEL
LIN {X 0,Y 431.906,Z 500.238,A -85,B 0,C 180,E1 -9340.018,E2 -9340.018} C_VEL
LIN {X 0,Y 432.049,Z 497.968,A -85,B 0,C 180,E1 -9342.974,E2 -9342.974} C_VEL
LIN {X 0,Y 432.145,Z 495.754,A -85,B 0,C 180,E1 -9345.88,E2 -9345.88} C_VEL
LIN {X 0,Y 432.273,Z 495.27,A -85,B 0,C 180,E1 -9347.287,E2 -9347.287} C_VEL
LIN {X 0,Y 432.437,Z 495.245,A -85,B 0,C 180,E1 -9350.646,E2 -9350.646} C_VEL
LIN {X 0,Y 432.57,Z 495.228,A -85,B 0,C 180,E1 -9353.469,E2 -9353.469} C_VEL
LIN {X 0,Y 432.401,Z 495.25,A -85,B 0,C 180,E1 -9355.338,E2 -9355.338} C_VEL
LIN {X 0,Y 432.602,Z 495.224,A -85,B 0,C 180,E1 -9358.138,E2 -9358.138} C_VEL
LIN {X 0,Y 432.73,Z 495.209,A -85,B 0,C 180,E1 -9360,E2 -9360} C_VEL
LIN {X 0,Y 432.602,Z 495.223,A -85,B 0,C 180,E1 -9362.793,E2 -9362.793} C_VEL
LIN {X 0,Y 432.571,Z 495.226,A -85,B 0,C 180,E1 -9366.53,E2 -9366.53} C_VEL
LIN {X 0,Y 432.44,Z 495.244,A -85,B 0,C 180,E1 -9369.353,E2 -9369.353} C_VEL
LIN {X 0,Y 432.427,Z 495.247,A -85,B 0,C 180,E1 -9372.803,E2 -9372.803} C_VEL
LIN {X 0,Y 432.409,Z 495.249,A -85,B 0,C 180,E1 -9376.479,E2 -9376.479} C_VEL
LIN {X 0,Y 432.335,Z 495.255,A -85,B 0,C 180,E1 -9379.96,E2 -9379.96} C_VEL
LIN {X 0,Y 432.316,Z 495.257,A -85,B 0,C 180,E1 -9382.964,E2 -9382.964} C_VEL
LIN {X 0,Y 432.361,Z 495.256,A -85,B 0,C 180,E1 -9386.032,E2 -9386.032} C_VEL
LIN {X 0,Y 432.349,Z 495.255,A -85,B 0,C 180,E1 -9389.187,E2 -9389.187} C_VEL
LIN {X 0,Y 432.323,Z 495.261,A -85,B 0,C 180,E1 -9392.293,E2 -9392.293} C_VEL
LIN {X 0,Y 432.338,Z 495.256,A -85,B 0,C 180,E1 -9394.677,E2 -9394.677} C_VEL
LIN {X 0,Y 432.342,Z 495.254,A -85,B 0,C 180,E1 -9398.149,E2 -9398.149} C_VEL
LIN {X 0,Y 432.377,Z 495.268,A -85,B 0,C 180,E1 -9399.981,E2 -9399.981} C_VEL
LIN {X 0,Y 433.127,Z 499.686,A -85,B 0,C 180,E1 -9403.099,E2 -9403.099} C_VEL
LIN {X 0,Y 433.928,Z 504.032,A -85,B 0,C 180,E1 -9405.858,E2 -9405.858} C_VEL
LIN {X 0,Y 434.373,Z 507.9,A -85,B 0,C 180,E1 -9408.095,E2 -9408.095} C_VEL
LIN {X 0,Y 434.01,Z 513.147,A -85,B 0,C 180,E1 -9410.837,E2 -9410.837} C_VEL
LIN {X 0,Y 433.537,Z 520.245,A -85,B 0,C 180,E1 -9414.297,E2 -9414.297} C_VEL
LIN {X 0,Y 433.092,Z 527.494,A -85,B 0,C 180,E1 -9417.622,E2 -9417.622} C_VEL
LIN {X 0,Y 432.663,Z 534.858,A -85,B 0,C 180,E1 -9420.836,E2 -9420.836} C_VEL
LIN {X 0,Y 432.343,Z 542.326,A -85,B 0,C 180,E1 -9423.966,E2 -9423.966} C_VEL
LIN {X 0,Y 432.112,Z 548.046,A -85,B 0,C 180,E1 -9426.283,E2 -9426.283} C_VEL
LIN {X 0,Y 436.192,Z 565.065,A -85,B 0,C 180,E1 -9426.927,E2 -9426.927} C_VEL
LIN {X 0,Y 439.068,Z 580.852,A -85,B 0,C 180,E1 -9427.666,E2 -9427.666} C_VEL
LIN {X 0,Y 439.818,Z 585.959,A -85,B 0,C 180,E1 -9427.941,E2 -9427.941} C_VEL
LIN {X 0,Y 438.952,Z 599.633,A -85,B 0,C 180,E1 -9428.639,E2 -9428.639} C_VEL
LIN {X 0,Y 437.904,Z 612.433,A -85,B 0,C 180,E1 -9429.447,E2 -9429.447} C_VEL
LIN {X 0,Y 436.759,Z 625.881,A -85,B 0,C 180,E1 -9430.495,E2 -9430.495} C_VEL
LIN {X 0,Y 435.569,Z 639.374,A -85,B 0,C 180,E1 -9431.783,E2 -9431.783} C_VEL
LIN {X 0,Y 434.631,Z 650.693,A -85,B 0,C 180,E1 -9433.078,E2 -9433.078} C_VEL
LIN {X 0,Y 433.654,Z 661.102,A -85,B 0,C 180,E1 -9434.49,E2 -9434.49} C_VEL
LIN {X 0,Y 432.84,Z 671.324,A -85,B 0,C 180,E1 -9436.143,E2 -9436.143} C_VEL
LIN {X 0,Y 432.188,Z 680.949,A -85,B 0,C 180,E1 -9438.034,E2 -9438.034} C_VEL
LIN {X 0,Y 431.717,Z 687.831,A -85,B 0,C 180,E1 -9439.684,E2 -9439.684} C_VEL
LIN {X 0,Y 431.466,Z 694.222,A -85,B 0,C 180,E1 -9441.57,E2 -9441.57} C_VEL
LIN {X 0,Y 431.331,Z 699.174,A -85,B 0,C 180,E1 -9443.45,E2 -9443.45} C_VEL
LIN {X 0,Y 431.235,Z 702.809,A -85,B 0,C 180,E1 -9445.326,E2 -9445.326} C_VEL
LIN {X 0,Y 431.283,Z 705.215,A -85,B 0,C 180,E1 -9447.197,E2 -9447.197} C_VEL
LIN {X 0,Y 431.286,Z 706.438,A -85,B 0,C 180,E1 -9449.066,E2 -9449.066} C_VEL
LIN {X 0,Y 431.286,Z 706.468,A -85,B 0,C 180,E1 -9450.933,E2 -9450.933} C_VEL
LIN {X 0,Y 431.28,Z 705.295,A -85,B 0,C 180,E1 -9452.802,E2 -9452.802} C_VEL
LIN {X 0,Y 431.234,Z 702.942,A -85,B 0,C 180,E1 -9454.673,E2 -9454.673} C_VEL
LIN {X 0,Y 431.369,Z 699.371,A -85,B 0,C 180,E1 -9456.548,E2 -9456.548} C_VEL
LIN {X 0,Y 431.473,Z 694.479,A -85,B 0,C 180,E1 -9458.429,E2 -9458.429} C_VEL
LIN {X 0,Y 431.717,Z 688.144,A -85,B 0,C 180,E1 -9460.315,E2 -9460.315} C_VEL
LIN {X 0,Y 432.187,Z 681.317,A -85,B 0,C 180,E1 -9461.965,E2 -9461.965} C_VEL
LIN {X 0,Y 432.846,Z 671.747,A -85,B 0,C 180,E1 -9463.856,E2 -9463.856} C_VEL
LIN {X 0,Y 433.673,Z 661.574,A -85,B 0,C 180,E1 -9465.509,E2 -9465.509} C_VEL
LIN {X 0,Y 434.682,Z 651.203,A -85,B 0,C 180,E1 -9466.919,E2 -9466.919} C_VEL
LIN {X 0,Y 435.706,Z 638.792,A -85,B 0,C 180,E1 -9468.332,E2 -9468.332} C_VEL
LIN {X 0,Y 436.851,Z 626.395,A -85,B 0,C 180,E1 -9469.5,E2 -9469.5} C_VEL
LIN {X 0,Y 437.912,Z 612.875,A -85,B 0,C 180,E1 -9470.552,E2 -9470.552} C_VEL
LIN {X 0,Y 439.099,Z 597.937,A -85,B 0,C 180,E1 -9471.476,E2 -9471.476} C_VEL
LIN {X 0,Y 439.862,Z 585.675,A -85,B 0,C 180,E1 -9472.073,E2 -9472.073} C_VEL
LIN {X 0,Y 437.019,Z 570.155,A -85,B 0,C 180,E1 -9472.832,E2 -9472.832} C_VEL
LIN {X 0,Y 433.475,Z 554.886,A -85,B 0,C 180,E1 -9473.433,E2 -9473.433} C_VEL
LIN {X 0,Y 432.192,Z 549.353,A -85,B 0,C 180,E1 -9473.628,E2 -9473.628} C_VEL
LIN {X 0,Y 432.563,Z 541.071,A -85,B 0,C 180,E1 -9477.059,E2 -9477.059} C_VEL
LIN {X 0,Y 433.016,Z 532.669,A -85,B 0,C 180,E1 -9480.66,E2 -9480.66} C_VEL
LIN {X 0,Y 433.387,Z 526.301,A -85,B 0,C 180,E1 -9483.459,E2 -9483.459} C_VEL
LIN {X 0,Y 433.807,Z 518.982,A -85,B 0,C 180,E1 -9486.827,E2 -9486.827} C_VEL
LIN {X 0,Y 434.296,Z 512.897,A -85,B 0,C 180,E1 -9489.731,E2 -9489.731} C_VEL
LIN {X 0,Y 434.518,Z 508.494,A -85,B 0,C 180,E1 -9491.926,E2 -9491.926} C_VEL
LIN {X 0,Y 433.888,Z 503.6,A -85,B 0,C 180,E1 -9494.545,E2 -9494.545} C_VEL
LIN {X 0,Y 432.896,Z 498.227,A -85,B 0,C 180,E1 -9497.643,E2 -9497.643} C_VEL
LIN {X 0,Y 432.382,Z 495.254,A -85,B 0,C 180,E1 -9499.446,E2 -9499.446} C_VEL
LIN {X 0,Y 432.326,Z 495.259,A -85,B 0,C 180,E1 -9502.8,E2 -9502.8} C_VEL
LIN {X 0,Y 432.351,Z 495.256,A -85,B 0,C 180,E1 -9505.996,E2 -9505.996} C_VEL
LIN {X 0,Y 432.386,Z 495.252,A -85,B 0,C 180,E1 -9509.744,E2 -9509.744} C_VEL
LIN {X 0,Y 432.39,Z 495.252,A -85,B 0,C 180,E1 -9513.372,E2 -9513.372} C_VEL
LIN {X 0,Y 432.361,Z 495.254,A -85,B 0,C 180,E1 -9516.023,E2 -9516.023} C_VEL
LIN {X 0,Y 432.34,Z 495.257,A -85,B 0,C 180,E1 -9519.046,E2 -9519.046} C_VEL
LIN {X 0,Y 432.368,Z 495.252,A -85,B 0,C 180,E1 -9522.011,E2 -9522.011} C_VEL
LIN {X 0,Y 432.391,Z 495.249,A -85,B 0,C 180,E1 -9524.927,E2 -9524.927} C_VEL
LIN {X 0,Y 432.471,Z 495.241,A -85,B 0,C 180,E1 -9527.804,E2 -9527.804} C_VEL
LIN {X 0,Y 432.482,Z 495.241,A -85,B 0,C 180,E1 -9531.59,E2 -9531.59} C_VEL
LIN {X 0,Y 432.591,Z 495.223,A -85,B 0,C 180,E1 -9534.406,E2 -9534.406} C_VEL
LIN {X 0,Y 432.596,Z 495.224,A -85,B 0,C 180,E1 -9538.138,E2 -9538.138} C_VEL
LIN {X 0,Y 432.725,Z 495.209,A -85,B 0,C 180,E1 -9540,E2 -9540} C_VEL
LIN {X 0,Y 432.599,Z 495.223,A -85,B 0,C 180,E1 -9542.794,E2 -9542.794} C_VEL
LIN {X 0,Y 432.567,Z 495.226,A -85,B 0,C 180,E1 -9546.531,E2 -9546.531} C_VEL
LIN {X 0,Y 432.434,Z 495.246,A -85,B 0,C 180,E1 -9549.354,E2 -9549.354} C_VEL
LIN {X 0,Y 432.421,Z 495.245,A -85,B 0,C 180,E1 -9552.804,E2 -9552.804} C_VEL
LIN {X 0,Y 432.404,Z 495.246,A -85,B 0,C 180,E1 -9556.48,E2 -9556.48} C_VEL
LIN {X 0,Y 432.331,Z 495.259,A -85,B 0,C 180,E1 -9559.961,E2 -9559.961} C_VEL
LIN {X 0,Y 432.312,Z 495.26,A -85,B 0,C 180,E1 -9562.965,E2 -9562.965} C_VEL
LIN {X 0,Y 432.357,Z 495.254,A -85,B 0,C 180,E1 -9566.033,E2 -9566.033} C_VEL
LIN {X 0,Y 432.346,Z 495.256,A -85,B 0,C 180,E1 -9569.188,E2 -9569.188} C_VEL
LIN {X 0,Y 432.326,Z 495.257,A -85,B 0,C 180,E1 -9572.296,E2 -9572.296} C_VEL
LIN {X 0,Y 432.335,Z 495.255,A -85,B 0,C 180,E1 -9574.678,E2 -9574.678} C_VEL
LIN {X 0,Y 432.349,Z 495.254,A -85,B 0,C 180,E1 -9578.149,E2 -9578.149} C_VEL
LIN {X 0,Y 432.369,Z 495.255,A -85,B 0,C 180,E1 -9581.609,E2 -9581.609} C_VEL
LIN {X 0,Y 432.375,Z 495.251,A -85,B 0,C 180,E1 -9584.343,E2 -9584.343} C_VEL
LIN {X 0,Y 432.363,Z 495.253,A -85,B 0,C 180,E1 -9587.01,E2 -9587.01} C_VEL
LIN {X 0,Y 432.357,Z 495.257,A -85,B 0,C 180,E1 -9589.818,E2 -9589.818} C_VEL
LIN {X 0,Y 432.316,Z 495.259,A -85,B 0,C 180,E1 -9593.024,E2 -9593.024} C_VEL
LIN {X 0,Y 432.359,Z 495.255,A -85,B 0,C 180,E1 -9595.998,E2 -9595.998} C_VEL
LIN {X 0,Y 432.348,Z 495.257,A -85,B 0,C 180,E1 -9599.491,E2 -9599.491} C_VEL
LIN {X 0,Y 432.394,Z 495.248,A -85,B 0,C 180,E1 -9602.93,E2 -9602.93} C_VEL
LIN {X 0,Y 432.374,Z 495.253,A -85,B 0,C 180,E1 -9606.025,E2 -9606.025} C_VEL
LIN {X 0,Y 432.353,Z 495.254,A -85,B 0,C 180,E1 -9609.047,E2 -9609.047} C_VEL
LIN {X 0,Y 432.382,Z 495.252,A -85,B 0,C 180,E1 -9612.012,E2 -9612.012} C_VEL
LIN {X 0,Y 432.399,Z 495.248,A -85,B 0,C 180,E1 -9614.927,E2 -9614.927} C_VEL
LIN {X 0,Y 432.463,Z 495.243,A -85,B 0,C 180,E1 -9617.804,E2 -9617.804} C_VEL
LIN {X 0,Y 432.468,Z 495.242,A -85,B 0,C 180,E1 -9621.59,E2 -9621.59} C_VEL
LIN {X 0,Y 432.602,Z 495.222,A -85,B 0,C 180,E1 -9624.407,E2 -9624.407} C_VEL
LIN {X 0,Y 432.612,Z 495.223,A -85,B 0,C 180,E1 -9628.139,E2 -9628.139} C_VEL
LIN {X 0,Y 432.737,Z 495.207,A -85,B 0,C 180,E1 -9630,E2 -9630} C_VEL
LIN {X 0,Y 432.376,Z 495.251,A -85,B 0,C 180,E1 -9632.795,E2 -9632.795} C_VEL
LIN {X 0,Y 432.119,Z 495.283,A -85,B 0,C 180,E1 -9635.03,E2 -9635.03} C_VEL
LIN {X 0,Y 431.372,Z 495.449,A -85,B 0,C 180,E1 -9635.807,E2 -9635.807} C_VEL
LIN {X 0,Y 428.402,Z 496.228,A -85,B 0,C 180,E1 -9637.064,E2 -9637.064} C_VEL
LIN {X 0,Y 425.919,Z 497.113,A -85,B 0,C 180,E1 -9638.076,E2 -9638.076} C_VEL
LIN {X 0,Y 424.851,Z 497.818,A -85,B 0,C 180,E1 -9638.859,E2 -9638.859} C_VEL
LIN {X 0,Y 424.762,Z 498.045,A -85,B 0,C 180,E1 -9639.125,E2 -9639.125} C_VEL
LIN {X 0,Y 424.679,Z 500.91,A -85,B 0,C 180,E1 -9642.473,E2 -9642.473} C_VEL
LIN {X 0,Y 424.573,Z 504.038,A -85,B 0,C 180,E1 -9646.044,E2 -9646.044} C_VEL
LIN {X 0,Y 427.791,Z 513.532,A -85,B 0,C 180,E1 -9646.482,E2 -9646.482} C_VEL
LIN {X 0,Y 432.446,Z 528.031,A -85,B 0,C 180,E1 -9647.239,E2 -9647.239} C_VEL
LIN {X 0,Y 433.95,Z 534.188,A -85,B 0,C 180,E1 -9647.586,E2 -9647.586} C_VEL
LIN {X 0,Y 433.128,Z 548.929,A -85,B 0,C 180,E1 -9648.324,E2 -9648.324} C_VEL
LIN {X 0,Y 432.088,Z 562.516,A -85,B 0,C 180,E1 -9649.187,E2 -9649.187} C_VEL
LIN {X 0,Y 430.955,Z 576.259,A -85,B 0,C 180,E1 -9650.276,E2 -9650.276} C_VEL
LIN {X 0,Y 429.881,Z 588.753,A -85,B 0,C 180,E1 -9651.489,E2 -9651.489} C_VEL
LIN {X 0,Y 428.601,Z 601.01,A -85,B 0,C 180,E1 -9652.92,E2 -9652.92} C_VEL
LIN {X 0,Y 427.536,Z 612.302,A -85,B 0,C 180,E1 -9654.524,E2 -9654.524} C_VEL
LIN {X 0,Y 426.587,Z 621.839,A -85,B 0,C 180,E1 -9656.149,E2 -9656.149} C_VEL
LIN {X 0,Y 425.851,Z 629.844,A -85,B 0,C 180,E1 -9657.789,E2 -9657.789} C_VEL
LIN {X 0,Y 425.208,Z 637.6,A -85,B 0,C 180,E1 -9659.726,E2 -9659.726} C_VEL
LIN {X 0,Y 424.787,Z 643,A -85,B 0,C 180,E1 -9661.41,E2 -9661.41} C_VEL
LIN {X 0,Y 424.49,Z 647.391,A -85,B 0,C 180,E1 -9663.117,E2 -9663.117} C_VEL
LIN {X 0,Y 424.345,Z 649.767,A -85,B 0,C 180,E1 -9664.271,E2 -9664.271} C_VEL
LIN {X 0,Y 424.178,Z 652.155,A -85,B 0,C 180,E1 -9665.721,E2 -9665.721} C_VEL
LIN {X 0,Y 424.048,Z 654.36,A -85,B 0,C 180,E1 -9667.823,E2 -9667.823} C_VEL
LIN {X 0,Y 424.005,Z 655.009,A -85,B 0,C 180,E1 -9669.04,E2 -9669.04} C_VEL
LIN {X 0,Y 423.982,Z 655.163,A -85,B 0,C 180,E1 -9670.314,E2 -9670.314} C_VEL
LIN {X 0,Y 424.01,Z 654.74,A -85,B 0,C 180,E1 -9671.765,E2 -9671.765} C_VEL
LIN {X 0,Y 424.115,Z 653.731,A -85,B 0,C 180,E1 -9673.186,E2 -9673.186} C_VEL
LIN {X 0,Y 424.331,Z 650.795,A -85,B 0,C 180,E1 -9675.413,E2 -9675.413} C_VEL
LIN {X 0,Y 424.59,Z 647.106,A -85,B 0,C 180,E1 -9677.261,E2 -9677.261} C_VEL
LIN {X 0,Y 424.902,Z 642.263,A -85,B 0,C 180,E1 -9679.087,E2 -9679.087} C_VEL
LIN {X 0,Y 425.495,Z 635.357,A -85,B 0,C 180,E1 -9681.122,E2 -9681.122} C_VEL
LIN {X 0,Y 426.224,Z 627.355,A -85,B 0,C 180,E1 -9682.997,E2 -9682.997} C_VEL
LIN {X 0,Y 427.044,Z 619.081,A -85,B 0,C 180,E1 -9684.59,E2 -9684.59} C_VEL
LIN {X 0,Y 427.991,Z 610.023,A -85,B 0,C 180,E1 -9686.06,E2 -9686.06} C_VEL
LIN {X 0,Y 429.091,Z 599.195,A -85,B 0,C 180,E1 -9687.54,E2 -9687.54} C_VEL
LIN {X 0,Y 430.299,Z 587.228,A -85,B 0,C 180,E1 -9688.9,E2 -9688.9} C_VEL
LIN {X 0,Y 431.369,Z 575.105,A -85,B 0,C 180,E1 -9690.05,E2 -9690.05} C_VEL
LIN {X 0,Y 432.494,Z 561.561,A -85,B 0,C 180,E1 -9691.101,E2 -9691.101} C_VEL
LIN {X 0,Y 433.534,Z 547.737,A -85,B 0,C 180,E1 -9691.958,E2 -9691.958} C_VEL
LIN {X 0,Y 434.177,Z 533.318,A -85,B 0,C 180,E1 -9692.666,E2 -9692.666} C_VEL
LIN {X 0,Y 429.574,Z 518.974,A -85,B 0,C 180,E1 -9693.5,E2 -9693.5} C_VEL
LIN {X 0,Y 424.686,Z 505.726,A -85,B 0,C 180,E1 -9694.186,E2 -9694.186} C_VEL
LIN {X 0,Y 424.819,Z 502.805,A -85,B 0,C 180,E1 -9697.885,E2 -9697.885} C_VEL
LIN {X 0,Y 424.929,Z 500.631,A -85,B 0,C 180,E1 -9700.683,E2 -9700.683} C_VEL
LIN {X 0,Y 425.064,Z 498.366,A -85,B 0,C 180,E1 -9703.675,E2 -9703.675} C_VEL
LIN {X 0,Y 425.154,Z 496.192,A -85,B 0,C 180,E1 -9706.618,E2 -9706.618} C_VEL
LIN {X 0,Y 425.343,Z 496.131,A -85,B 0,C 180,E1 -9709.528,E2 -9709.528} C_VEL
LIN {X 0,Y 425.535,Z 496.105,A -85,B 0,C 180,E1 -9712.407,E2 -9712.407} C_VEL
LIN {X 0,Y 425.552,Z 496.104,A -85,B 0,C 180,E1 -9714.313,E2 -9714.313} C_VEL
LIN {X 0,Y 425.572,Z 496.099,A -85,B 0,C 180,E1 -9718.107,E2 -9718.107} C_VEL
LIN {X 0,Y 425.699,Z 496.084,A -85,B 0,C 180,E1 -9720,E2 -9720} C_VEL
LIN {X 0,Y 425.554,Z 496.101,A -85,B 0,C 180,E1 -9722.84,E2 -9722.84} C_VEL
LIN {X 0,Y 425.529,Z 496.104,A -85,B 0,C 180,E1 -9726.639,E2 -9726.639} C_VEL
LIN {X 0,Y 425.398,Z 496.121,A -85,B 0,C 180,E1 -9729.509,E2 -9729.509} C_VEL
LIN {X 0,Y 425.39,Z 496.122,A -85,B 0,C 180,E1 -9732.903,E2 -9732.903} C_VEL
LIN {X 0,Y 425.358,Z 496.129,A -85,B 0,C 180,E1 -9736.605,E2 -9736.605} C_VEL
LIN {X 0,Y 425.325,Z 496.127,A -85,B 0,C 180,E1 -9739.636,E2 -9739.636} C_VEL
LIN {X 0,Y 425.304,Z 496.13,A -85,B 0,C 180,E1 -9743.365,E2 -9743.365} C_VEL
LIN {X 0,Y 425.345,Z 496.127,A -85,B 0,C 180,E1 -9746.844,E2 -9746.844} C_VEL
LIN {X 0,Y 425.315,Z 496.134,A -85,B 0,C 180,E1 -9749.717,E2 -9749.717} C_VEL
LIN {X 0,Y 425.279,Z 496.136,A -85,B 0,C 180,E1 -9753.048,E2 -9753.048} C_VEL
LIN {X 0,Y 425.282,Z 496.136,A -85,B 0,C 180,E1 -9755.929,E2 -9755.929} C_VEL
LIN {X 0,Y 425.354,Z 496.204,A -85,B 0,C 180,E1 -9759.536,E2 -9759.536} C_VEL
LIN {X 0,Y 426.035,Z 500.372,A -85,B 0,C 180,E1 -9762.559,E2 -9762.559} C_VEL
LIN {X 0,Y 426.723,Z 504.185,A -85,B 0,C 180,E1 -9765.088,E2 -9765.088} C_VEL
LIN {X 0,Y 427.346,Z 508.589,A -85,B 0,C 180,E1 -9767.736,E2 -9767.736} C_VEL
LIN {X 0,Y 427.151,Z 512.943,A -85,B 0,C 180,E1 -9770.083,E2 -9770.083} C_VEL
LIN {X 0,Y 426.588,Z 520.362,A -85,B 0,C 180,E1 -9773.83,E2 -9773.83} C_VEL
LIN {X 0,Y 426.221,Z 525.959,A -85,B 0,C 180,E1 -9776.469,E2 -9776.469} C_VEL
LIN {X 0,Y 425.751,Z 533.257,A -85,B 0,C 180,E1 -9779.77,E2 -9779.77} C_VEL
LIN {X 0,Y 425.338,Z 541.084,A -85,B 0,C 180,E1 -9783.158,E2 -9783.158} C_VEL
LIN {X 0,Y 425.044,Z 547.479,A -85,B 0,C 180,E1 -9785.833,E2 -9785.833} C_VEL
LIN {X 0,Y 429.671,Z 566.362,A -85,B 0,C 180,E1 -9786.597,E2 -9786.597} C_VEL
LIN {X 0,Y 432.522,Z 582.746,A -85,B 0,C 180,E1 -9787.405,E2 -9787.405} C_VEL
LIN {X 0,Y 433.11,Z 587.589,A -85,B 0,C 180,E1 -9787.673,E2 -9787.673} C_VEL
LIN {X 0,Y 432.144,Z 601.305,A -85,B 0,C 180,E1 -9788.411,E2 -9788.411} C_VEL
LIN {X 0,Y 430.93,Z 615.242,A -85,B 0,C 180,E1 -9789.349,E2 -9789.349} C_VEL
LIN {X 0,Y 429.729,Z 628.075,A -85,B 0,C 180,E1 -9790.411,E2 -9790.411} C_VEL
LIN {X 0,Y 428.639,Z 640.019,A -85,B 0,C 180,E1 -9791.601,E2 -9791.601} C_VEL
LIN {X 0,Y 427.584,Z 652.062,A -85,B 0,C 180,E1 -9793.037,E2 -9793.037} C_VEL
LIN {X 0,Y 426.586,Z 662.218,A -85,B 0,C 180,E1 -9794.471,E2 -9794.471} C_VEL
LIN {X 0,Y 425.733,Z 672.177,A -85,B 0,C 180,E1 -9796.151,E2 -9796.151} C_VEL
LIN {X 0,Y 425.161,Z 680.509,A -85,B 0,C 180,E1 -9797.833,E2 -9797.833} C_VEL
LIN {X 0,Y 424.688,Z 687.397,A -85,B 0,C 180,E1 -9799.511,E2 -9799.511} C_VEL
LIN {X 0,Y 424.395,Z 693.784,A -85,B 0,C 180,E1 -9801.428,E2 -9801.428} C_VEL
LIN {X 0,Y 424.242,Z 698.737,A -85,B 0,C 180,E1 -9803.341,E2 -9803.341} C_VEL
LIN {X 0,Y 424.163,Z 702.377,A -85,B 0,C 180,E1 -9805.247,E2 -9805.247} C_VEL
LIN {X 0,Y 424.214,Z 704.787,A -85,B 0,C 180,E1 -9807.151,E2 -9807.151} C_VEL
LIN {X 0,Y 424.198,Z 706.011,A -85,B 0,C 180,E1 -9809.05,E2 -9809.05} C_VEL
LIN {X 0,Y 424.198,Z 706.043,A -85,B 0,C 180,E1 -9810.949,E2 -9810.949} C_VEL
LIN {X 0,Y 424.211,Z 704.871,A -85,B 0,C 180,E1 -9812.848,E2 -9812.848} C_VEL
LIN {X 0,Y 424.163,Z 702.517,A -85,B 0,C 180,E1 -9814.752,E2 -9814.752} C_VEL
LIN {X 0,Y 424.291,Z 698.942,A -85,B 0,C 180,E1 -9816.658,E2 -9816.658} C_VEL
LIN {X 0,Y 424.401,Z 694.046,A -85,B 0,C 180,E1 -9818.571,E2 -9818.571} C_VEL
LIN {X 0,Y 424.688,Z 687.703,A -85,B 0,C 180,E1 -9820.488,E2 -9820.488} C_VEL
LIN {X 0,Y 425.164,Z 680.865,A -85,B 0,C 180,E1 -9822.166,E2 -9822.166} C_VEL
LIN {X 0,Y 425.737,Z 672.579,A -85,B 0,C 180,E1 -9823.848,E2 -9823.848} C_VEL
LIN {X 0,Y 426.603,Z 662.654,A -85,B 0,C 180,E1 -9825.527,E2 -9825.527} C_VEL
LIN {X 0,Y 427.631,Z 652.51,A -85,B 0,C 180,E1 -9826.96,E2 -9826.96} C_VEL
LIN {X 0,Y 428.671,Z 640.461,A -85,B 0,C 180,E1 -9828.396,E2 -9828.396} C_VEL
LIN {X 0,Y 429.81,Z 628.453,A -85,B 0,C 180,E1 -9829.584,E2 -9829.584} C_VEL
LIN {X 0,Y 430.936,Z 615.48,A -85,B 0,C 180,E1 -9830.65,E2 -9830.65} C_VEL
LIN {X 0,Y 432.145,Z 601.336,A -85,B 0,C 180,E1 -9831.588,E2 -9831.588} C_VEL
LIN {X 0,Y 433.144,Z 586.67,A -85,B 0,C 180,E1 -9832.354,E2 -9832.354} C_VEL
LIN {X 0,Y 430.329,Z 571.264,A -85,B 0,C 180,E1 -9833.143,E2 -9833.143} C_VEL
LIN {X 0,Y 426.868,Z 556.207,A -85,B 0,C 180,E1 -9833.769,E2 -9833.769} C_VEL
LIN {X 0,Y 425.196,Z 549.016,A -85,B 0,C 180,E1 -9834.02,E2 -9834.02} C_VEL
LIN {X 0,Y 425.585,Z 540.693,A -85,B 0,C 180,E1 -9837.54,E2 -9837.54} C_VEL
LIN {X 0,Y 425.982,Z 532.966,A -85,B 0,C 180,E1 -9840.917,E2 -9840.917} C_VEL
LIN {X 0,Y 426.429,Z 525.975,A -85,B 0,C 180,E1 -9844.079,E2 -9844.079} C_VEL
LIN {X 0,Y 426.985,Z 518.048,A -85,B 0,C 180,E1 -9847.809,E2 -9847.809} C_VEL
LIN {X 0,Y 427.494,Z 511.835,A -85,B 0,C 180,E1 -9850.867,E2 -9850.867} C_VEL
LIN {X 0,Y 427.36,Z 507.779,A -85,B 0,C 180,E1 -9852.997,E2 -9852.997} C_VEL
LIN {X 0,Y 426.723,Z 504.035,A -85,B 0,C 180,E1 -9855.087,E2 -9855.087} C_VEL
LIN {X 0,Y 425.673,Z 497.984,A -85,B 0,C 180,E1 -9858.669,E2 -9858.669} C_VEL
LIN {X 0,Y 425.334,Z 496.131,A -85,B 0,C 180,E1 -9859.878,E2 -9859.878} C_VEL
LIN {X 0,Y 425.263,Z 496.138,A -85,B 0,C 180,E1 -9863.492,E2 -9863.492} C_VEL
LIN {X 0,Y 425.299,Z 496.135,A -85,B 0,C 180,E1 -9865.817,E2 -9865.817} C_VEL
LIN {X 0,Y 425.291,Z 496.136,A -85,B 0,C 180,E1 -9869.236,E2 -9869.236} C_VEL
LIN {X 0,Y 425.341,Z 496.125,A -85,B 0,C 180,E1 -9872.442,E2 -9872.442} C_VEL
LIN {X 0,Y 425.341,Z 496.13,A -85,B 0,C 180,E1 -9875.602,E2 -9875.602} C_VEL
LIN {X 0,Y 425.283,Z 496.134,A -85,B 0,C 180,E1 -9878.681,E2 -9878.681} C_VEL
LIN {X 0,Y 425.323,Z 496.133,A -85,B 0,C 180,E1 -9881.703,E2 -9881.703} C_VEL
LIN {X 0,Y 425.345,Z 496.125,A -85,B 0,C 180,E1 -9884.671,E2 -9884.671} C_VEL
LIN {X 0,Y 425.42,Z 496.12,A -85,B 0,C 180,E1 -9887.599,E2 -9887.599} C_VEL
LIN {X 0,Y 425.433,Z 496.119,A -85,B 0,C 180,E1 -9891.45,E2 -9891.45} C_VEL
LIN {X 0,Y 425.547,Z 496.1,A -85,B 0,C 180,E1 -9894.314,E2 -9894.314} C_VEL
LIN {X 0,Y 425.566,Z 496.1,A -85,B 0,C 180,E1 -9898.108,E2 -9898.108} C_VEL
LIN {X 0,Y 425.694,Z 496.085,A -85,B 0,C 180,E1 -9900,E2 -9900} C_VEL
LIN {X 0,Y 425.551,Z 496.101,A -85,B 0,C 180,E1 -9902.84,E2 -9902.84} C_VEL
LIN {X 0,Y 425.57,Z 496.102,A -85,B 0,C 180,E1 -9905.687,E2 -9905.687} C_VEL
LIN {X 0,Y 425.433,Z 496.115,A -85,B 0,C 180,E1 -9908.551,E2 -9908.551} C_VEL
LIN {X 0,Y 425.403,Z 496.119,A -85,B 0,C 180,E1 -9912.402,E2 -9912.402} C_VEL
LIN {X 0,Y 425.379,Z 496.121,A -85,B 0,C 180,E1 -9916.313,E2 -9916.313} C_VEL
LIN {X 0,Y 425.32,Z 496.133,A -85,B 0,C 180,E1 -9919.637,E2 -9919.637} C_VEL
LIN {X 0,Y 425.299,Z 496.135,A -85,B 0,C 180,E1 -9923.366,E2 -9923.366} C_VEL
LIN {X 0,Y 425.342,Z 496.126,A -85,B 0,C 180,E1 -9926.846,E2 -9926.846} C_VEL
LIN {X 0,Y 425.312,Z 496.134,A -85,B 0,C 180,E1 -9929.718,E2 -9929.718} C_VEL
LIN {X 0,Y 425.278,Z 496.136,A -85,B 0,C 180,E1 -9933.049,E2 -9933.049} C_VEL
LIN {X 0,Y 425.28,Z 496.136,A -85,B 0,C 180,E1 -9935.93,E2 -9935.93} C_VEL
LIN {X 0,Y 425.31,Z 496.131,A -85,B 0,C 180,E1 -9939.048,E2 -9939.048} C_VEL
LIN {X 0,Y 425.328,Z 496.128,A -85,B 0,C 180,E1 -9942.647,E2 -9942.647} C_VEL
LIN {X 0,Y 425.316,Z 496.131,A -85,B 0,C 180,E1 -9946.053,E2 -9946.053} C_VEL
LIN {X 0,Y 425.308,Z 496.13,A -85,B 0,C 180,E1 -9948.627,E2 -9948.627} C_VEL
LIN {X 0,Y 425.323,Z 496.13,A -85,B 0,C 180,E1 -9951.106,E2 -9951.106} C_VEL
LIN {X 0,Y 425.3,Z 496.131,A -85,B 0,C 180,E1 -9954.665,E2 -9954.665} C_VEL
LIN {X 0,Y 425.265,Z 496.137,A -85,B 0,C 180,E1 -9958.074,E2 -9958.074} C_VEL
LIN {X 0,Y 425.332,Z 496.131,A -85,B 0,C 180,E1 -9961.369,E2 -9961.369} C_VEL
LIN {X 0,Y 425.297,Z 496.132,A -85,B 0,C 180,E1 -9964.556,E2 -9964.556} C_VEL
LIN {X 0,Y 425.29,Z 496.137,A -85,B 0,C 180,E1 -9967.662,E2 -9967.662} C_VEL
LIN {X 0,Y 425.365,Z 496.123,A -85,B 0,C 180,E1 -9970.705,E2 -9970.705} C_VEL
LIN {X 0,Y 425.392,Z 496.124,A -85,B 0,C 180,E1 -9973.689,E2 -9973.689} C_VEL
LIN {X 0,Y 425.416,Z 496.122,A -85,B 0,C 180,E1 -9977.599,E2 -9977.599} C_VEL
LIN {X 0,Y 425.412,Z 496.121,A -85,B 0,C 180,E1 -9981.45,E2 -9981.45} C_VEL
LIN {X 0,Y 425.557,Z 496.1,A -85,B 0,C 180,E1 -9984.314,E2 -9984.314} C_VEL
LIN {X 0,Y 425.582,Z 496.098,A -85,B 0,C 180,E1 -9988.108,E2 -9988.108} C_VEL
LIN {X 0,Y 425.707,Z 496.083,A -85,B 0,C 180,E1 -9990,E2 -9990} C_VEL
LIN {X 0,Y 425.311,Z 496.131,A -85,B 0,C 180,E1 -9992.842,E2 -9992.842} C_VEL
LIN {X 0,Y 425.027,Z 496.17,A -85,B 0,C 180,E1 -9995.694,E2 -9995.694} C_VEL
LIN {X 0,Y 424.89,Z 496.282,A -85,B 0,C 180,E1 -9997.043,E2 -9997.043} C_VEL
LIN {X 0,Y 424.762,Z 498.045,A -85,B 0,C 180,E1 -9999.125,E2 -9999.125} C_VEL
LIN {X 0,Y 424.078,Z 498.783,A -85,B 0,C 180,E1 -9999.91,E2 -9999.91} C_VEL
LIN {X 0,Y 421.179,Z 500.193,A -85,B 0,C 180,E1 -10001.182,E2 -10001.182} C_VEL
LIN {X 0,Y 418.723,Z 501.346,A -85,B 0,C 180,E1 -10002.208,E2 -10002.208} C_VEL
LIN {X 0,Y 417.662,Z 502.15,A -85,B 0,C 180,E1 -10003.003,E2 -10003.003} C_VEL
LIN {X 0,Y 417.571,Z 502.391,A -85,B 0,C 180,E1 -10003.273,E2 -10003.273} C_VEL
LIN {X 0,Y 417.502,Z 504.456,A -85,B 0,C 180,E1 -10005.649,E2 -10005.649} C_VEL
LIN {X 0,Y 421.723,Z 516.665,A -85,B 0,C 180,E1 -10006.221,E2 -10006.221} C_VEL
LIN {X 0,Y 426.337,Z 531.383,A -85,B 0,C 180,E1 -10007.037,E2 -10007.037} C_VEL
LIN {X 0,Y 427.227,Z 534.516,A -85,B 0,C 180,E1 -10007.224,E2 -10007.224} C_VEL
LIN {X 0,Y 426.503,Z 549.541,A -85,B 0,C 180,E1 -10007.997,E2 -10007.997} C_VEL
LIN {X 0,Y 425.375,Z 563.727,A -85,B 0,C 180,E1 -10008.92,E2 -10008.92} C_VEL
LIN {X 0,Y 424.244,Z 576.831,A -85,B 0,C 180,E1 -10009.98,E2 -10009.98} C_VEL
LIN {X 0,Y 423.145,Z 588.971,A -85,B 0,C 180,E1 -10011.177,E2 -10011.177} C_VEL
LIN {X 0,Y 421.886,Z 600.47,A -85,B 0,C 180,E1 -10012.529,E2 -10012.529} C_VEL
LIN {X 0,Y 420.893,Z 610.159,A -85,B 0,C 180,E1 -10013.886,E2 -10013.886} C_VEL
LIN {X 0,Y 419.896,Z 620.052,A -85,B 0,C 180,E1 -10015.529,E2 -10015.529} C_VEL
LIN {X 0,Y 419.004,Z 628.699,A -85,B 0,C 180,E1 -10017.254,E2 -10017.254} C_VEL
LIN {X 0,Y 418.322,Z 636.51,A -85,B 0,C 180,E1 -10019.158,E2 -10019.158} C_VEL
LIN {X 0,Y 417.816,Z 642.384,A -85,B 0,C 180,E1 -10020.922,E2 -10020.922} C_VEL
LIN {X 0,Y 417.492,Z 647.084,A -85,B 0,C 180,E1 -10022.68,E2 -10022.68} C_VEL
LIN {X 0,Y 417.247,Z 650.54,A -85,B 0,C 180,E1 -10024.376,E2 -10024.376} C_VEL
LIN {X 0,Y 417.055,Z 653.173,A -85,B 0,C 180,E1 -10026.143,E2 -10026.143} C_VEL
LIN {X 0,Y 416.959,Z 654.628,A -85,B 0,C 180,E1 -10027.607,E2 -10027.607} C_VEL
LIN {X 0,Y 416.902,Z 655.586,A -85,B 0,C 180,E1 -10029.836,E2 -10029.836} C_VEL
LIN {X 0,Y 416.91,Z 655.482,A -85,B 0,C 180,E1 -10031.104,E2 -10031.104} C_VEL
LIN {X 0,Y 416.971,Z 654.84,A -85,B 0,C 180,E1 -10032.391,E2 -10032.391} C_VEL
LIN {X 0,Y 417.056,Z 653.67,A -85,B 0,C 180,E1 -10033.702,E2 -10033.702} C_VEL
LIN {X 0,Y 417.289,Z 650.922,A -85,B 0,C 180,E1 -10035.683,E2 -10035.683} C_VEL
LIN {X 0,Y 417.589,Z 646.629,A -85,B 0,C 180,E1 -10037.775,E2 -10037.775} C_VEL
LIN {X 0,Y 417.987,Z 641.205,A -85,B 0,C 180,E1 -10039.745,E2 -10039.745} C_VEL
LIN {X 0,Y 418.621,Z 634.734,A -85,B 0,C 180,E1 -10041.598,E2 -10041.598} C_VEL
LIN {X 0,Y 419.31,Z 627.674,A -85,B 0,C 180,E1 -10043.251,E2 -10043.251} C_VEL
LIN {X 0,Y 420.331,Z 618.026,A -85,B 0,C 180,E1 -10045.117,E2 -10045.117} C_VEL
LIN {X 0,Y 421.473,Z 607.698,A -85,B 0,C 180,E1 -10046.757,E2 -10046.757} C_VEL
LIN {X 0,Y 422.692,Z 596.524,A -85,B 0,C 180,E1 -10048.231,E2 -10048.231} C_VEL
LIN {X 0,Y 423.916,Z 584.508,A -85,B 0,C 180,E1 -10049.552,E2 -10049.552} C_VEL
LIN {X 0,Y 425.134,Z 571.652,A -85,B 0,C 180,E1 -10050.719,E2 -10050.719} C_VEL
LIN {X 0,Y 426.296,Z 557.357,A -85,B 0,C 180,E1 -10051.774,E2 -10051.774} C_VEL
LIN {X 0,Y 427.385,Z 542.653,A -85,B 0,C 180,E1 -10052.62,E2 -10052.62} C_VEL
LIN {X 0,Y 427.744,Z 535.42,A -85,B 0,C 180,E1 -10052.966,E2 -10052.966} C_VEL
LIN {X 0,Y 423.344,Z 521.461,A -85,B 0,C 180,E1 -10053.818,E2 -10053.818} C_VEL
LIN {X 0,Y 417.773,Z 506.832,A -85,B 0,C 180,E1 -10054.597,E2 -10054.597} C_VEL
LIN {X 0,Y 417.673,Z 506.211,A -85,B 0,C 180,E1 -10054.657,E2 -10054.657} C_VEL
LIN {X 0,Y 417.788,Z 503.394,A -85,B 0,C 180,E1 -10058.279,E2 -10058.279} C_VEL
LIN {X 0,Y 417.892,Z 501.056,A -85,B 0,C 180,E1 -10061.365,E2 -10061.365} C_VEL
LIN {X 0,Y 418.016,Z 498.776,A -85,B 0,C 180,E1 -10064.395,E2 -10064.395} C_VEL
LIN {X 0,Y 418.174,Z 497.026,A -85,B 0,C 180,E1 -10067.1,E2 -10067.1} C_VEL
LIN {X 0,Y 418.332,Z 497.004,A -85,B 0,C 180,E1 -10070.328,E2 -10070.328} C_VEL
LIN {X 0,Y 418.49,Z 496.981,A -85,B 0,C 180,E1 -10073.249,E2 -10073.249} C_VEL
LIN {X 0,Y 418.34,Z 497.001,A -85,B 0,C 180,E1 -10075.181,E2 -10075.181} C_VEL
LIN {X 0,Y 418.542,Z 496.975,A -85,B 0,C 180,E1 -10078.075,E2 -10078.075} C_VEL
LIN {X 0,Y 418.669,Z 496.96,A -85,B 0,C 180,E1 -10080,E2 -10080} C_VEL
LIN {X 0,Y 418.507,Z 496.98,A -85,B 0,C 180,E1 -10082.887,E2 -10082.887} C_VEL
LIN {X 0,Y 418.491,Z 496.982,A -85,B 0,C 180,E1 -10086.751,E2 -10086.751} C_VEL
LIN {X 0,Y 418.338,Z 497,A -85,B 0,C 180,E1 -10089.671,E2 -10089.671} C_VEL
LIN {X 0,Y 418.343,Z 496.999,A -85,B 0,C 180,E1 -10093,E2 -10093} C_VEL
LIN {X 0,Y 418.309,Z 497.005,A -85,B 0,C 180,E1 -10096.735,E2 -10096.735} C_VEL
LIN {X 0,Y 418.267,Z 497.006,A -85,B 0,C 180,E1 -10099.79,E2 -10099.79} C_VEL
LIN {X 0,Y 418.235,Z 497.012,A -85,B 0,C 180,E1 -10102.736,E2 -10102.736} C_VEL
LIN {X 0,Y 418.268,Z 497.01,A -85,B 0,C 180,E1 -10105.904,E2 -10105.904} C_VEL
LIN {X 0,Y 418.271,Z 497.009,A -85,B 0,C 180,E1 -10109.161,E2 -10109.161} C_VEL
LIN {X 0,Y 418.255,Z 497.011,A -85,B 0,C 180,E1 -10112.844,E2 -10112.844} C_VEL
LIN {X 0,Y 418.246,Z 497.013,A -85,B 0,C 180,E1 -10116.239,E2 -10116.239} C_VEL
LIN {X 0,Y 418.268,Z 497.148,A -85,B 0,C 180,E1 -10119.051,E2 -10119.051} C_VEL
LIN {X 0,Y 418.969,Z 501.236,A -85,B 0,C 180,E1 -10122.142,E2 -10122.142} C_VEL
LIN {X 0,Y 419.828,Z 505.957,A -85,B 0,C 180,E1 -10125.325,E2 -10125.325} C_VEL
LIN {X 0,Y 420.348,Z 509.285,A -85,B 0,C 180,E1 -10127.362,E2 -10127.362} C_VEL
LIN {X 0,Y 420.261,Z 512.688,A -85,B 0,C 180,E1 -10129.293,E2 -10129.293} C_VEL
LIN {X 0,Y 419.726,Z 518.639,A -85,B 0,C 180,E1 -10132.408,E2 -10132.408} C_VEL
LIN {X 0,Y 419.363,Z 524.409,A -85,B 0,C 180,E1 -10135.264,E2 -10135.264} C_VEL
LIN {X 0,Y 418.852,Z 532.05,A -85,B 0,C 180,E1 -10138.841,E2 -10138.841} C_VEL
LIN {X 0,Y 418.398,Z 539.018,A -85,B 0,C 180,E1 -10141.944,E2 -10141.944} C_VEL
LIN {X 0,Y 418.041,Z 546.436,A -85,B 0,C 180,E1 -10145.147,E2 -10145.147} C_VEL
LIN {X 0,Y 418.02,Z 546.977,A -85,B 0,C 180,E1 -10145.375,E2 -10145.375} C_VEL
LIN {X 0,Y 422.552,Z 565.036,A -85,B 0,C 180,E1 -10146.134,E2 -10146.134} C_VEL
LIN {X 0,Y 425.153,Z 579.523,A -85,B 0,C 180,E1 -10146.855,E2 -10146.855} C_VEL
LIN {X 0,Y 426.467,Z 588.161,A -85,B 0,C 180,E1 -10147.347,E2 -10147.347} C_VEL
LIN {X 0,Y 425.353,Z 602.971,A -85,B 0,C 180,E1 -10148.176,E2 -10148.176} C_VEL
LIN {X 0,Y 424.129,Z 616.479,A -85,B 0,C 180,E1 -10149.129,E2 -10149.129} C_VEL
LIN {X 0,Y 422.775,Z 630.306,A -85,B 0,C 180,E1 -10150.328,E2 -10150.328} C_VEL
LIN {X 0,Y 421.629,Z 641.795,A -85,B 0,C 180,E1 -10151.536,E2 -10151.536} C_VEL
LIN {X 0,Y 420.525,Z 653.458,A -85,B 0,C 180,E1 -10152.994,E2 -10152.994} C_VEL
LIN {X 0,Y 419.527,Z 663.301,A -85,B 0,C 180,E1 -10154.452,E2 -10154.452} C_VEL
LIN {X 0,Y 418.651,Z 672.997,A -85,B 0,C 180,E1 -10156.159,E2 -10156.159} C_VEL
LIN {X 0,Y 418.062,Z 681.104,A -85,B 0,C 180,E1 -10157.869,E2 -10157.869} C_VEL
LIN {X 0,Y 417.511,Z 688.682,A -85,B 0,C 180,E1 -10159.819,E2 -10159.819} C_VEL
LIN {X 0,Y 417.281,Z 694.716,A -85,B 0,C 180,E1 -10161.769,E2 -10161.769} C_VEL
LIN {X 0,Y 417.123,Z 699.446,A -85,B 0,C 180,E1 -10163.759,E2 -10163.759} C_VEL
LIN {X 0,Y 417.091,Z 701.949,A -85,B 0,C 180,E1 -10165.167,E2 -10165.167} C_VEL
LIN {X 0,Y 417.128,Z 704.36,A -85,B 0,C 180,E1 -10167.102,E2 -10167.102} C_VEL
LIN {X 0,Y 417.114,Z 705.584,A -85,B 0,C 180,E1 -10169.034,E2 -10169.034} C_VEL
LIN {X 0,Y 417.114,Z 705.617,A -85,B 0,C 180,E1 -10170.965,E2 -10170.965} C_VEL
LIN {X 0,Y 417.123,Z 704.442,A -85,B 0,C 180,E1 -10172.897,E2 -10172.897} C_VEL
LIN {X 0,Y 417.093,Z 702.084,A -85,B 0,C 180,E1 -10174.832,E2 -10174.832} C_VEL
LIN {X 0,Y 417.222,Z 698.502,A -85,B 0,C 180,E1 -10176.771,E2 -10176.771} C_VEL
LIN {X 0,Y 417.317,Z 693.593,A -85,B 0,C 180,E1 -10178.717,E2 -10178.717} C_VEL
LIN {X 0,Y 417.662,Z 687.243,A -85,B 0,C 180,E1 -10180.666,E2 -10180.666} C_VEL
LIN {X 0,Y 418.139,Z 679.266,A -85,B 0,C 180,E1 -10182.62,E2 -10182.62} C_VEL
LIN {X 0,Y 418.913,Z 670.791,A -85,B 0,C 180,E1 -10184.326,E2 -10184.326} C_VEL
LIN {X 0,Y 419.814,Z 660.579,A -85,B 0,C 180,E1 -10186.034,E2 -10186.034} C_VEL
LIN {X 0,Y 420.916,Z 650.181,A -85,B 0,C 180,E1 -10187.489,E2 -10187.489} C_VEL
LIN {X 0,Y 422.099,Z 637.73,A -85,B 0,C 180,E1 -10188.945,E2 -10188.945} C_VEL
LIN {X 0,Y 423.358,Z 625.302,A -85,B 0,C 180,E1 -10190.148,E2 -10190.148} C_VEL
LIN {X 0,Y 424.553,Z 611.737,A -85,B 0,C 180,E1 -10191.229,E2 -10191.229} C_VEL
LIN {X 0,Y 425.806,Z 596.695,A -85,B 0,C 180,E1 -10192.181,E2 -10192.181} C_VEL
LIN {X 0,Y 426.368,Z 586.99,A -85,B 0,C 180,E1 -10192.681,E2 -10192.681} C_VEL
LIN {X 0,Y 423.45,Z 571.272,A -85,B 0,C 180,E1 -10193.511,E2 -10193.511} C_VEL
LIN {X 0,Y 419.848,Z 555.725,A -85,B 0,C 180,E1 -10194.174,E2 -10194.174} C_VEL
LIN {X 0,Y 418.121,Z 548.61,A -85,B 0,C 180,E1 -10194.432,E2 -10194.432} C_VEL
LIN {X 0,Y 418.529,Z 541.474,A -85,B 0,C 180,E1 -10197.525,E2 -10197.525} C_VEL
LIN {X 0,Y 418.962,Z 533.274,A -85,B 0,C 180,E1 -10201.184,E2 -10201.184} C_VEL
LIN {X 0,Y 419.41,Z 526.818,A -85,B 0,C 180,E1 -10204.148,E2 -10204.148} C_VEL
LIN {X 0,Y 420.041,Z 518.495,A -85,B 0,C 180,E1 -10208.151,E2 -10208.151} C_VEL
LIN {X 0,Y 420.539,Z 512.371,A -85,B 0,C 180,E1 -10211.233,E2 -10211.233} C_VEL
LIN {X 0,Y 420.313,Z 508.58,A -85,B 0,C 180,E1 -10213.278,E2 -10213.278} C_VEL
LIN {X 0,Y 419.323,Z 502.827,A -85,B 0,C 180,E1 -10216.593,E2 -10216.593} C_VEL
LIN {X 0,Y 418.29,Z 497.009,A -85,B 0,C 180,E1 -10220.225,E2 -10220.225} C_VEL
LIN {X 0,Y 418.238,Z 497.013,A -85,B 0,C 180,E1 -10223.976,E2 -10223.976} C_VEL
LIN {X 0,Y 418.249,Z 497.013,A -85,B 0,C 180,E1 -10227.155,E2 -10227.155} C_VEL
LIN {X 0,Y 418.265,Z 497.008,A -85,B 0,C 180,E1 -10230.838,E2 -10230.838} C_VEL
LIN {X 0,Y 418.261,Z 497.009,A -85,B 0,C 180,E1 -10234.096,E2 -10234.096} C_VEL
LIN {X 0,Y 418.222,Z 497.016,A -85,B 0,C 180,E1 -10237.263,E2 -10237.263} C_VEL
LIN {X 0,Y 418.273,Z 497.006,A -85,B 0,C 180,E1 -10240.364,E2 -10240.364} C_VEL
LIN {X 0,Y 418.316,Z 497.005,A -85,B 0,C 180,E1 -10243.405,E2 -10243.405} C_VEL
LIN {X 0,Y 418.345,Z 496.999,A -85,B 0,C 180,E1 -10246.994,E2 -10246.994} C_VEL
LIN {X 0,Y 418.351,Z 496.997,A -85,B 0,C 180,E1 -10250.329,E2 -10250.329} C_VEL
LIN {X 0,Y 418.485,Z 496.984,A -85,B 0,C 180,E1 -10253.249,E2 -10253.249} C_VEL
LIN {X 0,Y 418.336,Z 497.001,A -85,B 0,C 180,E1 -10255.182,E2 -10255.182} C_VEL
LIN {X 0,Y 418.535,Z 496.975,A -85,B 0,C 180,E1 -10258.076,E2 -10258.076} C_VEL
LIN {X 0,Y 418.664,Z 496.96,A -85,B 0,C 180,E1 -10260,E2 -10260} C_VEL
LIN {X 0,Y 418.505,Z 496.978,A -85,B 0,C 180,E1 -10262.888,E2 -10262.888} C_VEL
LIN {X 0,Y 418.484,Z 496.98,A -85,B 0,C 180,E1 -10266.597,E2 -10266.597} C_VEL
LIN {X 0,Y 418.333,Z 497.003,A -85,B 0,C 180,E1 -10269.672,E2 -10269.672} C_VEL
LIN {X 0,Y 418.337,Z 497,A -85,B 0,C 180,E1 -10273.001,E2 -10273.001} C_VEL
LIN {X 0,Y 418.304,Z 497.002,A -85,B 0,C 180,E1 -10276.736,E2 -10276.736} C_VEL
LIN {X 0,Y 418.262,Z 497.012,A -85,B 0,C 180,E1 -10279.791,E2 -10279.791} C_VEL
LIN {X 0,Y 418.23,Z 497.012,A -85,B 0,C 180,E1 -10282.737,E2 -10282.737} C_VEL
LIN {X 0,Y 418.264,Z 497.01,A -85,B 0,C 180,E1 -10285.905,E2 -10285.905} C_VEL
LIN {X 0,Y 418.268,Z 497.009,A -85,B 0,C 180,E1 -10289.162,E2 -10289.162} C_VEL
LIN {X 0,Y 418.254,Z 497.009,A -85,B 0,C 180,E1 -10292.846,E2 -10292.846} C_VEL
LIN {X 0,Y 418.244,Z 497.011,A -85,B 0,C 180,E1 -10296.24,E2 -10296.24} C_VEL
LIN {X 0,Y 418.263,Z 497.012,A -85,B 0,C 180,E1 -10299.681,E2 -10299.681} C_VEL
LIN {X 0,Y 418.281,Z 497.006,A -85,B 0,C 180,E1 -10302.331,E2 -10302.331} C_VEL
LIN {X 0,Y 418.271,Z 497.009,A -85,B 0,C 180,E1 -10305.115,E2 -10305.115} C_VEL
